FUNCTION_BLOCK UInterface EXTENDS OperationalParticleSet
  VAR CONSTANT
    cStartPeriod : t_ms_time := TIME#2s0ms;
  END_VAR
  VAR
    lVROverrideRadioReady : ValueReferenceBool;
    lOverrideRadioReady : BOOL := FALSE;
    lAlarmUInterfaceEstop : ReportableSystemControl;
    lAlarmUInterfaceStop : ReportableSystemControl;
    lAlarmUInterfaceEmgy : ReportableSystemControl;
    lAlarmUInterfaceNotReady : ReportableSystemControl;
    lUInterfaceId : t_ui_id := t_ui_id.cUIIdNone;
    lResolved : REFERENCE TO UInterface;
    lSingleMode : BOOL := TRUE;
    lUIMode : t_ui_mode := cUIModeInoperable;
    lUIModeRequest : BOOL := FALSE;
    lReady : BOOL := FALSE;
    lDiagnostic : t_uinterface_diagnostic;
    _Diagnostic : t_uinterface_diagnostic;
  END_VAR

            ;
          

METHOD operator
                  lDiagnostic := _Diagnostic;
_Diagnostic := cUInterfaceDiagnosticOK;

SUPER^.operator();

(* events for radios that are not present are ignored if in multi mode *)
IF (lSingleMode) THEN
	lUIMode := cUIModeSingle;
END_IF

IF ((NOT(Estop)) AND (lUIMode>cUIModeInoperable)) THEN
	Diagnostic := cUInterfaceDiagnosticEstop;

	lAlarmUInterfaceEstop.trigger(FALSE);
END_IF

IF ((NOT(Stop)) AND (lUIMode>cUIModeInoperable)) THEN
	Diagnostic := cUInterfaceDiagnosticStop;

	lAlarmUInterfaceStop.trigger(FALSE);
END_IF

IF ((NOT(Emgy)) AND (lUIMode>cUIModeInoperable))  THEN
	Diagnostic := cUInterfaceDiagnosticEmgy;

	lAlarmUInterfaceEmgy.trigger(FALSE);
END_IF

lReady := ((Stop) AND (Emgy) AND (Estop));
IF (NOT(Ready)) THEN
	lUIMode := cUIModeInoperable;

	IF (lSingleMode) THEN
		Diagnostic := cUInterfaceDiagnosticNotReady;
	
		lAlarmUInterfaceNotReady.trigger(FALSE);
	END_IF
END_IF

IF (UIModeResponse) THEN
	Resolved.uiModeHandler(UInterfaceId);
END_IF

IF (lUIMode=cUIModeInoperable) THEN
	Diagnostic := cUInterfaceDiagnosticInoperable;
	RETURN;
END_IF

IF (lUIMode<cUIModeMaster) THEN
	Diagnostic := cUInterfaceDiagnosticNotMaster;
	RETURN;
END_IF


                
END_METHOD

METHOD uiModeHandler
  VAR_INPUT
    id : t_ui_id;
  END_VAR
                  
                
END_METHOD

METHOD initialize
                  lResolved REF= THIS^;

lVROverrideRadioReady.initializeValueReference(lOverrideRadioReady,NopSelf,'OvrdReady','Override UI to be ready','',cValueStyleParameter);

lAlarmUInterfaceEstop.initializeState(NopSelf,'',cACUInterfaceEstop); // foobar life was zero
lAlarmUInterfaceEstop.Control := cSystemControlStop;
lAlarmUInterfaceEstop.AllowableSystemState := cSystemStateCharging;

lAlarmUInterfaceStop.initializeState(NopSelf,'',cACUInterfaceStop);
lAlarmUInterfaceStop.Control := cSystemControlStop;
lAlarmUInterfaceStop.AllowableSystemState := cSystemStateCharging;
		
lAlarmUInterfaceEmgy.initializeState(NopSelf,'',cACUInterfaceEmgy);
lAlarmUInterfaceEmgy.Control := cSystemControlStop;
lAlarmUInterfaceEmgy.AllowableSystemState := cSystemStateCharging;

lAlarmUInterfaceNotReady.initializeState(NopSelf,'',cACUInterfaceNotReady);
lAlarmUInterfaceNotReady.Control := cSystemControlStop;
lAlarmUInterfaceNotReady.AllowableSystemState := cSystemStateCharging;

SUPER^.initialize();
SubSystem := cSubsystemUInterface;

lReady := FALSE;
lUIMode := cUIModeInoperable;
//lInputMode := cInputModeDefault;
                
END_METHOD

PROPERTY LiftBalanceAB : t_percentage
GET
                    LiftBalanceAB := 0;
                  
END_GET
END_PROPERTY

PROPERTY LiftBalanceAD : t_percentage
GET
                    LiftBalanceAD := 0;
                  
END_GET
END_PROPERTY

(* {attribute 'monitoring' := 'call'} *)
PROPERTY LiftJoystickInputPresent : BOOL
GET
                    LiftJoystickInputPresent := false;

                  
END_GET
END_PROPERTY

PROPERTY OperatingMethodRequest : t_operating_method
GET
                    OperatingMethodRequest := cOperatingMethodNone;

                  
END_GET
END_PROPERTY

PROPERTY Override : BOOL
GET
                    Override := false;
                  
END_GET
END_PROPERTY

PROPERTY Present : BOOL
GET
                    Present := (UIMode>t_ui_mode.cUIModeInoperable);

                  
END_GET
END_PROPERTY

(* {attribute 'monitoring' := 'call'} *)
PROPERTY Ready : BOOL
GET
                    Ready := ((lReady) OR (lOverrideRadioReady));

                  
END_GET
END_PROPERTY

PROPERTY SideshiftAB : t_percentage
GET
                    SideshiftAB := 0;

                  
END_GET
END_PROPERTY

PROPERTY SideshiftCD : t_percentage
GET
                    SideshiftCD := 0;

                  
END_GET
END_PROPERTY

PROPERTY SingleMode : BOOL
GET
                    SingleMode := lSingleMode;
                  
END_GET
SET
                    lSingleMode := SingleMode;
                  
END_SET
END_PROPERTY

PROPERTY SlowFactor : REAL
GET
                    SlowFactor := 1.0;

                  
END_GET
END_PROPERTY

PROPERTY SpreaderTelescopingExtend : BOOL
GET
                    SpreaderTelescopingExtend := FALSE;

                  
END_GET
END_PROPERTY

PROPERTY SpreaderTelescopingRetract : BOOL
GET
                    SpreaderTelescopingRetract := FALSE;

                  
END_GET
END_PROPERTY

PROPERTY Steer : t_percentage
GET
                    Steer := 0;
                  
END_GET
END_PROPERTY

PROPERTY SteerModeRequest : t_steer_mode
GET
                    SteerModeRequest := cSteerModeNone;

                  
END_GET
END_PROPERTY

PROPERTY Stop : BOOL
GET
                    Stop := true;
                  
END_GET
END_PROPERTY

PROPERTY Topbeam : t_percentage
GET
                    Topbeam := 0;
                  
END_GET
END_PROPERTY

(* {attribute 'monitoring' := 'call'} *)
PROPERTY Travel : t_percentage
GET
                    Travel := 0;
                  
END_GET
END_PROPERTY

(* {attribute 'monitoring' := 'call'} *)
PROPERTY TravelJoystickInputPresent : BOOL
GET
                    TravelJoystickInputPresent := false;

                  
END_GET
END_PROPERTY

PROPERTY TwistlockLock : BOOL
GET
                    TwistlockLock := false;
                  
END_GET
END_PROPERTY

PROPERTY TwistlockUnlock : BOOL
GET
                    TwistlockUnlock := false;
                  
END_GET
END_PROPERTY

PROPERTY TypeToken : t_medium_string
GET
                    TypeToken := 'UInterface';
                  
END_GET
END_PROPERTY

PROPERTY UIEventCodeRequest : t_ui_event_code
GET
                    UIEventCodeRequest := cUIEventCodeNone;
                  
END_GET
END_PROPERTY

(* {attribute 'monitoring' := 'call'} *)
PROPERTY UIMode : t_ui_mode
GET
                    UIMode := lUIMode;

                  
END_GET
SET
                    lUIMode := UIMode;
                  
END_SET
END_PROPERTY

(* {attribute 'monitoring' := 'call'} *)
PROPERTY UIModeRequest : BOOL
GET
                    UIModeRequest := lUIModeRequest;
                  
END_GET
SET
                    lUIModeRequest := UIModeRequest;
                  
END_SET
END_PROPERTY

(* {attribute 'monitoring' := 'call'} *)
PROPERTY UIModeResponse : BOOL
GET
                    UIModeResponse := FALSE;


                  
END_GET
END_PROPERTY

PROPERTY UInterfaceId : t_ui_id
GET
                    UInterfaceId := lUInterfaceId;
                  
END_GET
SET
                    lUInterfaceId := UInterfaceId;
                  
END_SET
END_PROPERTY

PROPERTY UIOrientation : t_ui_orientation
GET
                    UIOrientation := cUIOrientationForward;
                  
END_GET
END_PROPERTY

PROPERTY UMFS : BOOL
GET
                    UMFS := true;
                  
END_GET
END_PROPERTY

PROPERTY ZeroSteerTargetAngle : BOOL
GET
                    ZeroSteerTargetAngle := false;
                  
END_GET
END_PROPERTY

PROPERTY Resolved : REFERENCE TO UInterface
GET
                    Resolved ref= lResolved;
                  
END_GET
SET
                    lResolved ref= Resolved;
                  
END_SET
END_PROPERTY

PROPERTY Active : BOOL
GET
                    Active := (UIMode>cUIModeSlave);

                  
END_GET
END_PROPERTY

PROPERTY AutomationRequest : t_prog_mov_code
GET
                    AutomationRequest := cProgMovCodeNone;
                  
END_GET
END_PROPERTY

PROPERTY AutomationStart : BOOL
GET
                    AutomationStart := FALSE;

                  
END_GET
END_PROPERTY

(* {attribute 'monitoring' := 'call'} *)
PROPERTY ConfigurationJoystickInputPresent : BOOL
GET
                    ConfigurationJoystickInputPresent := FALSE;

                  
END_GET
END_PROPERTY

PROPERTY Diagnostic : t_uinterface_diagnostic
GET
                    Diagnostic := lDiagnostic;
                  
END_GET
SET
                    _Diagnostic := Diagnostic;
                  
END_SET
END_PROPERTY

PROPERTY Emgy : BOOL
GET
                    Emgy := true;
                  
END_GET
END_PROPERTY

PROPERTY Estop : BOOL
GET
                    Estop := true;
                  
END_GET
END_PROPERTY

PROPERTY FunctionalModeRequest : t_functional_mode
GET
                    FunctionalModeRequest := cFunctionalModeAny;

                  
END_GET
END_PROPERTY

PROPERTY Horn : BOOL
GET
                    Horn := false;
                  
END_GET
END_PROPERTY

PROPERTY InputMode : t_input_mode
GET
                    InputMode := cInputModeDefault;

                  
END_GET
END_PROPERTY

PROPERTY IsBeginner : BOOL
GET
                    IsBeginner := FALSE;

                  
END_GET
END_PROPERTY

PROPERTY IsSlow : BOOL
GET
                    IsSlow := FALSE;

                  
END_GET
END_PROPERTY

(* {attribute 'monitoring' := 'call'} *)
PROPERTY JoystickInputPresent : BOOL
GET
                    JoystickInputPresent := false;
                  
END_GET
END_PROPERTY

PROPERTY Lift : t_percentage
GET
                    Lift := 0;
                  
END_GET
END_PROPERTY

PROPERTY EnableBatteryPack : BOOL
GET
                    EnableBatteryPack := FALSE;

                  
END_GET
END_PROPERTY
END_FUNCTION_BLOCK

FUNCTION_BLOCK ExtractTest
  VAR
    mWordA : WORD;
    mWordB : WORD;
    mWordC : WORD;
    mWordD : WORD;
    mBoolA : BOOL;
    mBoolB : BOOL;
    mBoolC : BOOL;
    mIntA : INT;
    mIntB : INT;
    mIntC : INT;
    mIntD : INT;
    mByteA : BYTE;
    mByteB : BYTE;
    mByteC : BYTE;
    mByteD : BYTE;
    mStartA : USINT := 0;
    mStartB : USINT := 0;
    mStartC : USINT := 0;
    mStartD : USINT := 0;
    mStartE : USINT := 0;
    mStartF : USINT := 0;
    mLengthA : USINT := 0;
    mLengthB : USINT := 0;
  END_VAR

            mByteA := fInsertBool(pData:=mBoolA,pStart:=mStartA);
mByteB := fInsertBits(pData:=mIntA,pStart:=mStartB);
mByteC := fMergeBits(pByte:=mByteA,pData:=mIntB,pStart:=mStartC);

mWordA := fInsertBoolIntoWord(pData:=mBoolA,pStart:=mStartD);
mWordB := fInsertBitsIntoWord(pData:=mIntA,pStart:=mStartE);
mWordC := fMergeBitsIntoWord(pWord:=mWordA,pData:=mIntB,pStart:=mStartF);

mBoolB := fExtractBool(pByte:=mByteA,pStart:=mStartA);
mBoolC := fExtractBoolFromWord(pWord:=mWordA,pStart:=mStartD);

mIntC := fExtractBits(pByte:=mByteB,pStart:=mStartB,pLength:=mLengthA);
mIntD := fExtractBitsFromWord(pWord:=mWordB,pStart:=mStartE,pLength:=mLengthB);

mWordD :=  fExtractWord(pByte1:=mByteA ,pByte2:=mByteB);
          
END_FUNCTION_BLOCK

FUNCTION fExtractBits : INT
  VAR_INPUT
    pByte : BYTE;
    pStart : USINT;
    pLength : USINT;
  END_VAR

            fExtractBits := SHR(SHL(pByte,8-pStart-pLength),8-pLength);
          
END_FUNCTION

FUNCTION fExtractBitsFromWord : INT
  VAR_INPUT
    pWord : WORD;
    pStart : USINT;
    pLength : USINT;
  END_VAR

            fExtractBitsFromWord := WORD_TO_INT(SHR(SHL(pWord,16-pStart-pLength),16-pLength));
          
END_FUNCTION

FUNCTION fExtractBool : BOOL
  VAR_INPUT
    pByte : BYTE;
    pStart : USINT;
  END_VAR

            fExtractBool := BYTE_TO_BOOL(pByte AND SHL(BOOL_TO_BYTE(TRUE),pStart));
          
END_FUNCTION

FUNCTION fExtractBoolFromWord : BOOL
  VAR_INPUT
    pWord : WORD;
    pStart : USINT;
  END_VAR

            fExtractBoolFromWord := WORD_TO_BOOL(pWord AND SHL(BOOL_TO_WORD(TRUE),pStart));
          
END_FUNCTION

FUNCTION fExtractWord : WORD
  VAR_INPUT
    pByte1 : BYTE;
    pByte2 : BYTE;
  END_VAR

            fExtractWord := SHL(BYTE_TO_WORD(pByte2),8) OR BYTE_TO_WORD(pByte1);
          
END_FUNCTION

FUNCTION fInsertBits : BYTE
  VAR_INPUT
    pData : INT;
    pStart : USINT;
  END_VAR

            fInsertBits := SHL(INT_TO_BYTE(pData),pStart);
          
END_FUNCTION

FUNCTION fInsertBitsIntoWord : WORD
  VAR_INPUT
    pData : INT;
    pStart : USINT;
  END_VAR

            fInsertBitsIntoWord := SHL(INT_TO_WORD(pData),pStart);
          
END_FUNCTION

FUNCTION fInsertBool : BYTE
  VAR_INPUT
    pData : BOOL;
    pStart : USINT;
  END_VAR

            fInsertBool := SHL(BOOL_TO_BYTE(pData),pStart);
          
END_FUNCTION

FUNCTION fInsertBoolIntoWord : WORD
  VAR_INPUT
    pData : BOOL;
    pStart : USINT;
  END_VAR

            fInsertBoolIntoWord := SHL(BOOL_TO_WORD(pData),pStart);
          
END_FUNCTION

FUNCTION fMergeBits : BYTE
  VAR_INPUT
    pByte : BYTE;
    pData : INT;
    pStart : USINT;
  END_VAR

            fMergeBits := SHL(INT_TO_BYTE(pData),pStart) OR (pByte);
          
END_FUNCTION

FUNCTION fMergeBitsIntoBytes : WORD
  VAR_INPUT
    pByte1 : BYTE;
    pByte2 : BYTE;
    pData : INT;
    pStart : USINT;
  END_VAR

            fMergeBitsIntoBytes := SHL(INT_TO_WORD(pData),pStart) OR (SHL(BYTE_TO_WORD(pByte2),8) OR BYTE_TO_WORD(pByte1));
          
END_FUNCTION

FUNCTION fMergeBitsIntoWord : WORD
  VAR_INPUT
    pWord : WORD;
    pData : INT;
    pStart : USINT;
  END_VAR

            fMergeBitsIntoWord := SHL(INT_TO_WORD(pData),pStart) OR (pWord);
          
END_FUNCTION

FUNCTION fMergeBool : BYTE
  VAR_INPUT
    pByte : BYTE;
    pData : BOOL;
    pStart : USINT;
  END_VAR

            fMergeBool := SHL(BOOL_TO_BYTE(pData),pStart) OR (pByte);
          
END_FUNCTION

FUNCTION fMergeBoolIntoWord : WORD
  VAR_INPUT
    pWord : WORD;
    pData : BOOL;
    pStart : USINT;
  END_VAR

            fMergeBoolIntoWord := SHL(BOOL_TO_WORD(pData),pStart) OR (pWord);
          
END_FUNCTION

FUNCTION_BLOCK ValueObjectBoolChange EXTENDS ValueObjectBool
  VAR
    lPreviousValue : BOOL;
    lRising : BOOL := FALSE;
    lFalling : BOOL := FALSE;
  END_VAR

            
          

METHOD operator
                  SUPER^.operator();

lFalling := ((NOT(Value)) AND (lPreviousValue));
lRising := ((Value) AND (NOT(lPreviousValue)));

lPreviousValue := Value;

                
END_METHOD

(* {attribute 'monitoring' := 'call'} *)
PROPERTY Falling : BOOL
GET
                    Falling := lFalling;
                  
END_GET
END_PROPERTY

(* {attribute 'monitoring' := 'call'} *)
PROPERTY Rising : BOOL
GET
                    Rising := lRising;
                  
END_GET
END_PROPERTY
END_FUNCTION_BLOCK

FUNCTION_BLOCK ValueObjectBoolCheckReferenceDINT EXTENDS ValueObjectBool
  VAR
    lCheckReference : REFERENCE TO DINT;
    _CheckReference : DINT;
    lTimer : t_timer;
    lCheckRequiredValue : BOOL := TRUE;
    lCheckEnable : BOOL := TRUE;
    lCheckCritical : BOOL := FALSE;
    lError : BOOL := FALSE;
    lPrevious : BOOL;
    lChanged : BOOL;
    lOK : BOOL;
    lOKOff : BOOL;
    lOff : BOOL;
  END_VAR

            
          

METHOD initialize
                  IF (NOT(__ISVALIDREF(lCheckReference))) THEN
	lCheckReference REF= _CheckReference;
END_IF

_CheckReference := 0;

SUPER^.initialize();

lTimer.initialize();
lTimer.Enable := true;

lValue := lPrevious := lError := lOK := lOKOff := lOff := lChanged := FALSE;

                
END_METHOD

METHOD operator
                  IF (lPrevious<>lValue) THEN
	lChanged := TRUE;
	lPrevious := lValue;
	lTimer.reset();
ELSE
	lChanged := FALSE;
END_IF

SUPER^.operator();

lTimer.operator();

lError := ((lTimer.lExpired) AND
	(lValue) AND
	(lCheckEnable) AND
	(DINT_TO_BOOL(lCheckReference)<>lCheckRequiredValue));	

(* waits to set OK until timer has expired *)
lOK :=  ((lTimer.lExpired) AND (lValue) AND (NOT(lError)));
lOKOff :=  ((lTimer.lExpired) AND (NOT(lValue)) AND (NOT(lError)));
lOff := ((lTimer.lExpired) AND (NOT(lValue)));


                
END_METHOD

PROPERTY CheckCritical : BOOL
GET
                    CheckCritical := lCheckCritical;
                  
END_GET
SET
                    lCheckCritical := CheckCritical;
                  
END_SET
END_PROPERTY

PROPERTY CheckEnable : BOOL
GET
                    CheckEnable := lCheckEnable;
                  
END_GET
SET
                    lCheckEnable := CheckEnable;
                  
END_SET
END_PROPERTY

PROPERTY CheckPeriod : t_time
GET
                    CheckPeriod := lTimer.Period;
                  
END_GET
SET
                    lTimer.Period := CheckPeriod;

                  
END_SET
END_PROPERTY

PROPERTY Error : BOOL
GET
                    Error := lError;
                  
END_GET
END_PROPERTY

PROPERTY IsOff : BOOL
GET
                    IsOff := lOff;
                  
END_GET
END_PROPERTY

PROPERTY OK : BOOL
GET
                    OK := lOK;
                  
END_GET
END_PROPERTY

PROPERTY OKOff : BOOL
GET
                    OKOff := lOKOff;
                  
END_GET
END_PROPERTY

PROPERTY CheckReference : REFERENCE TO DINT
SET
                    lCheckReference Ref= CheckReference;
                  
END_SET
END_PROPERTY
END_FUNCTION_BLOCK

FUNCTION_BLOCK ValueObjectBoolCheckReferenceDINTOutputReferenceDINT EXTENDS ValueObjectBoolCheckReferenceDINT
  VAR
    lOutputReference : REFERENCE TO DINT;
  END_VAR

            
          

METHOD operator
                  SUPER^.operator();

lOutputReference := BOOL_TO_DINT(lValue);
                
END_METHOD

METHOD initialize
                  IF (NOT(__ISVALIDREF(lOutputReference))) THEN
	gCodeErrorHandler(pMessage:=CONCAT('null reference in ',lIdentity));
END_IF

SUPER^.initialize();

                
END_METHOD

PROPERTY OutputReference : REFERENCE TO DINT
SET
                    lOutputReference ref= OutputReference;
                  
END_SET
END_PROPERTY
END_FUNCTION_BLOCK

FUNCTION_BLOCK ValueObjectBoolInputRealThreshold EXTENDS ValueObjectBool
  VAR
    lInput : REAL;
    lBelowIsOn : BOOL;
    lThresholdOn : REAL;
    lThresholdOff : REAL;
    lHysteresis : REAL := 2.0;
    lThreshold : REAL := 30.0;
  END_VAR

            
          

METHOD operator
                  IF (lBelowIsOn) THEN
	// generally lThresholdBelowIsOn (off->on) < lThresholdLowerOff (on->off)
	IF ((lInput<=lThresholdOn) OR
		((lValue) AND (lInput<=lThresholdOff))) THEN
		lValue := TRUE;
	ELSE
		lValue := FALSE;
	END_IF
ELSE
	// generally lThresholdUpperOn (off->on) > lThresholdUpperOff (on->off)
	IF ((lInput>=lThresholdOn) OR
		((lValue) AND (lInput>=lThresholdOff))) THEN
		lValue := TRUE;
	ELSE
		lValue := FALSE;
	END_IF
END_IF

SUPER^.operator();


                
END_METHOD

METHOD describe
  VAR_INPUT
    executeContext : POINTER TO ExecuteContext;
  END_VAR
                  SUPER^.describe(executeContext);

IF (executeContext^.matchOption(cExecuteOptionSyntax)) THEN
	executeContext^.describeSyntaxConfigurable(lStyle,cTokenThreshold,cDataTypeReal,cEnumTypeNone,lUnits,cDescriptionThreshold);
	executeContext^.describeSyntaxConfigurable(lStyle,cTokenHysteresis,cDataTypeReal,cEnumTypeNone,lUnits,cDescriptionHysteresis);
	
	RETURN;
END_IF

IF (executeContext^.matchOption(cExecuteOptionParameter)) THEN
	executeContext^.describeParameter(lStyle,lIdentity,cTokenThreshold,gTypeHandler.getTokenForReal(lThreshold),cDataTypeReal,cEnumTypeNone,lUnits,cDescriptionThreshold);
	executeContext^.describeParameter(cValueStyleParameter,lIdentity,cTokenHysteresis,gTypeHandler.getTokenForReal(lHysteresis),cDataTypeReal,cEnumTypeNone,lUnits,cDescriptionHysteresis);
		
	RETURN;
END_IF

executeContext^.appendTokenPair(cTokenThreshold,gTypeHandler.getTokenForReal(lThreshold),FALSE,TRUE);
executeContext^.appendTokenPair(cTokenHysteresis,gTypeHandler.getTokenForReal(lHysteresis),FALSE,TRUE);
executeContext^.appendTokenPair(cTokenHysteresis,gTypeHandler.getTokenForUSINT(BOOL_TO_USINT(lBelowIsOn)),FALSE,TRUE);




                
END_METHOD

METHOD configure
  VAR_INPUT
    executeContext : POINTER TO ExecuteContext;
  END_VAR
                  IF (executeContext^.configureReal(cTokenThreshold,lThreshold,FALSE,THIS)) THEN
	RETURN;
END_IF

IF (executeContext^.configureReal(cTokenHysteresis,lHysteresis,FALSE,THIS)) THEN
	RETURN;
END_IF

SUPER^.configure(executeContext);


                
END_METHOD

METHOD setThresholds : BOOL
                  IF (lBelowIsOn) THEN
	lThresholdOff := Threshold + lHysteresis;
	lThresholdOn := Threshold - lHysteresis;
ELSE
	lThresholdOff := Threshold - lHysteresis;
	lThresholdOn := Threshold + lHysteresis;	
END_IF
                
END_METHOD

METHOD initialize
                  SUPER^.initialize();

setThresholds();
                
END_METHOD

PROPERTY Input : REAL
SET
                    lInput := Input;
operator();

                  
END_SET
END_PROPERTY

PROPERTY ThresholdOff : REAL
GET
                    ThresholdOff := lThresholdOff;
                  
END_GET
END_PROPERTY

PROPERTY ThresholdOn : REAL
GET
                    ThresholdOn := ThresholdOn;
                  
END_GET
END_PROPERTY

PROPERTY Hysteresis : REAL
GET
                    Hysteresis := lHysteresis;
                  
END_GET
SET
                    IF (lHysteresis=Hysteresis) THEN
	RETURN;
END_IF

lHysteresis := Hysteresis;
setThresholds();
                  
END_SET
END_PROPERTY

PROPERTY Threshold : REAL
GET
                    Threshold := lThreshold;
                  
END_GET
SET
                    IF (lThreshold=Threshold) THEN
	RETURN;
END_IF

lThreshold := Threshold;
setThresholds();
                  
END_SET
END_PROPERTY

PROPERTY BelowIsOn : BOOL
GET
                    BelowIsOn := lBelowIsOn;
                  
END_GET
SET
                    lBelowIsOn := BelowIsOn;
setThresholds();

                  
END_SET
END_PROPERTY
END_FUNCTION_BLOCK

FUNCTION_BLOCK ValueObjectBoolInputReferenceBool EXTENDS ValueObjectBool
  VAR
    lInputReference : REFERENCE TO BOOL;
  END_VAR

            
          

METHOD initialize
                  IF (NOT(__ISVALIDREF(lInputReference))) THEN
	gCodeErrorHandler(pMessage:=CONCAT('null reference in ',lIdentity));
END_IF

SUPER^.initialize();

                
END_METHOD

METHOD operator
                  lValue := lInputReference;

SUPER^.operator();

                
END_METHOD

PROPERTY InputReference : REFERENCE TO BOOL
SET
                    lInputReference REF= InputReference;


                  
END_SET
END_PROPERTY
END_FUNCTION_BLOCK

FUNCTION_BLOCK ValueObjectBoolInputReferenceBoolAndBool EXTENDS ValueObjectBool
  VAR
    lInputReferenceA : REFERENCE TO BOOL;
    lInputReferenceB : REFERENCE TO BOOL;
  END_VAR

            
          

METHOD initialize
                  IF ((NOT(__ISVALIDREF(lInputReferenceA))) OR
	(NOT(__ISVALIDREF(lInputReferenceB)))) THEN
	gCodeErrorHandler(pMessage:=CONCAT('null reference in ',lIdentity));
END_IF

SUPER^.initialize();

                
END_METHOD

METHOD operator
                  lValue := ((lInputReferenceA) AND (lInputReferenceB));

SUPER^.operator();

                
END_METHOD

PROPERTY InputReferenceA : REFERENCE TO BOOL
SET
                    lInputReferenceA REF= InputReferenceA;


                  
END_SET
END_PROPERTY

PROPERTY InputReferenceB : REFERENCE TO BOOL
SET
                    lInputReferenceB REF= InputReferenceB;


                  
END_SET
END_PROPERTY
END_FUNCTION_BLOCK

FUNCTION_BLOCK ValueObjectBoolInputReferenceBoolChange EXTENDS ValueObjectBool
  VAR
    lInputReference : REFERENCE TO BOOL;
    lPreviousValue : BOOL;
    lRising : BOOL := FALSE;
    lFalling : BOOL := FALSE;
  END_VAR

            
          

METHOD operator
                  lValue := lInputReference;

SUPER^.operator();

lFalling := ((NOT(Value)) AND (lPreviousValue));
lRising := ((Value) AND (NOT(lPreviousValue)));

lPreviousValue := Value;

                
END_METHOD

METHOD initialize
                  IF (NOT(__ISVALIDREF(lInputReference))) THEN
	gCodeErrorHandler(pMessage:=CONCAT('null reference in ',lIdentity));
END_IF

SUPER^.initialize();

                
END_METHOD

(* {attribute 'monitoring' := 'call'} *)
PROPERTY Falling : BOOL
GET
                    Falling := lFalling;
                  
END_GET
END_PROPERTY

(* {attribute 'monitoring' := 'call'} *)
PROPERTY Rising : BOOL
GET
                    Rising := lRising;
                  
END_GET
END_PROPERTY

PROPERTY InputReference : REFERENCE TO BOOL
SET
                    lInputReference REF= InputReference;


                  
END_SET
END_PROPERTY
END_FUNCTION_BLOCK

FUNCTION_BLOCK ValueObjectBoolInputReferenceDINTAsBool EXTENDS ValueObjectBool
  VAR
    lInputReference : REFERENCE TO DINT;
  END_VAR

            
          

METHOD initialize
                  IF (NOT(__ISVALIDREF(lInputReference))) THEN
	gCodeErrorHandler(pMessage:=CONCAT('null reference in ',lIdentity));
END_IF

SUPER^.initialize();

                
END_METHOD

METHOD operator
                  lValue := DINT_TO_BOOL(lInputReference);

SUPER^.operator();

                
END_METHOD

PROPERTY InputReference : REFERENCE TO DINT
SET
                    lInputReference REF= InputReference;


                  
END_SET
END_PROPERTY
END_FUNCTION_BLOCK

FUNCTION_BLOCK ValueObjectBoolInputReferenceDINTFiltered EXTENDS ValueObjectBool
  VAR
    lInputReference : REFERENCE TO DINT;
    lFilterEnabled : BOOL := TRUE;
    lPrevious : BOOL;
    lTimer : t_timer;
  END_VAR

            
          

METHOD initialize
                  IF (NOT(__ISVALIDREF(lInputReference))) THEN
	gCodeErrorHandler(pMessage:=CONCAT('null reference in ',lIdentity));
END_IF

SUPER^.initialize();

lTimer.initialize();
lTimer.Enable := TRUE;
lTImer.Period := T#100MS;

lPrevious := lValue;

                
END_METHOD

METHOD operator
                  IF (lFilterEnabled) THEN
	IF (lPrevious<>DINT_TO_BOOL(lInputReference)) THEN
		lTimer.reset();
	END_IF

	lTimer.operator();
	IF (lTimer.Expired) THEN
		lValue := DINT_TO_BOOL(lInputReference);
	END_IF
ELSE
	lValue := DINT_TO_BOOL(lInputReference);
END_IF

lPrevious := DINT_TO_BOOL(lInputReference);

SUPER^.operator();

                
END_METHOD

PROPERTY FilterEnabled : BOOL
GET
                    FilterEnabled := lFilterEnabled;
                  
END_GET
SET
                    lFilterEnabled := FilterEnabled;
                  
END_SET
END_PROPERTY

PROPERTY Period : t_time
GET
                    Period := lTimer.Period;
                  
END_GET
SET
                    lTimer.Period := Period;
                  
END_SET
END_PROPERTY

PROPERTY InputReference : REFERENCE TO DINT
SET
                    lInputReference REF= InputReference;


                  
END_SET
END_PROPERTY
END_FUNCTION_BLOCK

FUNCTION_BLOCK ValueObjectBoolInputReferenceUINT EXTENDS ValueObjectBool
  VAR
    lInputReference : REFERENCE TO UINT;
    lIndex : USINT;
  END_VAR

            
          

METHOD initialize
                  IF (NOT(__ISVALIDREF(lInputReference))) THEN
	gCodeErrorHandler(pMessage:=CONCAT('null reference in ',lIdentity));
END_IF

SUPER^.initialize();

                
END_METHOD

METHOD operator
                  lValue := fExtractBoolFromWord(UINT_TO_WORD(lInputReference),pStart:=lIndex);

SUPER^.operator();

                
END_METHOD

PROPERTY Index : USINT
GET
                    Index := lIndex;
                  
END_GET
SET
                    lIndex := MIN(Index,15);
                  
END_SET
END_PROPERTY

PROPERTY InputReference : REFERENCE TO UINT
SET
                    lInputReference REF= InputReference;


                  
END_SET
END_PROPERTY
END_FUNCTION_BLOCK

FUNCTION_BLOCK ValueObjectBoolInputReferenceUSINT EXTENDS ValueObjectBool
  VAR
    lInputReference : REFERENCE TO USINT;
    lIndex : USINT;
  END_VAR

            
          

METHOD initialize
                  IF (NOT(__ISVALIDREF(lInputReference))) THEN
	gCodeErrorHandler(pMessage:=CONCAT('null reference in ',lIdentity));
END_IF

SUPER^.initialize();

                
END_METHOD

METHOD operator
                  lValue := fExtractBoolFromWord(USINT_TO_WORD(lInputReference),pStart:=lIndex);

SUPER^.operator();

                
END_METHOD

PROPERTY Index : USINT
GET
                    Index := lIndex;
                  
END_GET
SET
                    lIndex := MIN(Index,7);
                  
END_SET
END_PROPERTY

PROPERTY InputReference : REFERENCE TO USINT
SET
                    lInputReference REF= InputReference;


                  
END_SET
END_PROPERTY
END_FUNCTION_BLOCK

FUNCTION_BLOCK ValueObjectBoolInputReferenceUSINTAsBool EXTENDS ValueObjectBool
  VAR
    lInputReference : REFERENCE TO USINT;
  END_VAR

            
          

METHOD initialize
                  IF (NOT(__ISVALIDREF(lInputReference))) THEN
	gCodeErrorHandler(pMessage:=CONCAT('null reference in ',lIdentity));
END_IF

SUPER^.initialize();

                
END_METHOD

METHOD operator
                  lValue := USINT_TO_BOOL(lInputReference);

SUPER^.operator();

                
END_METHOD

PROPERTY InputReference : REFERENCE TO USINT
SET
                    lInputReference REF= InputReference;


                  
END_SET
END_PROPERTY
END_FUNCTION_BLOCK

FUNCTION_BLOCK ValueObjectBoolInputReferenceUSINTChange EXTENDS ValueObjectBoolChange
  VAR
    lInputReference : REFERENCE TO USINT;
    lIndex : USINT;
  END_VAR

            
          

METHOD operator
                  lValue := fExtractBoolFromWord(USINT_TO_WORD(lInputReference),pStart:=lIndex);

SUPER^.operator();

lPreviousValue := Value;

                
END_METHOD

METHOD initialize
                  IF (NOT(__ISVALIDREF(lInputReference))) THEN
	gCodeErrorHandler(pMessage:=CONCAT('null reference in ',lIdentity));
END_IF

SUPER^.initialize();

                
END_METHOD

PROPERTY InputReference : REFERENCE TO USINT
SET
                    lInputReference REF= InputReference;


                  
END_SET
END_PROPERTY

PROPERTY Index : USINT
GET
                    Index := lIndex;
                  
END_GET
SET
                    lIndex := MIN(Index,7);
                  
END_SET
END_PROPERTY
END_FUNCTION_BLOCK

FUNCTION_BLOCK ValueObjectBoolLatch EXTENDS ValueObjectBoolChange

            
          

METHOD reset
                  lValue := FALSE;
operator();
                
END_METHOD

PROPERTY Input : BOOL
SET
                    IF (Input) THEN
	lValue := Input;
END_IF

operator();

                  
END_SET
END_PROPERTY
END_FUNCTION_BLOCK

FUNCTION_BLOCK ValueObjectBoolOutputReferenceBool EXTENDS ValueObjectBool
  VAR
    lOutputReference : REFERENCE TO BOOL;
  END_VAR

            
          

METHOD operator
                  SUPER^.operator();

lOutputReference := lValue;


                
END_METHOD

METHOD initialize
                  IF (NOT(__ISVALIDREF(lOutputReference))) THEN
	gCodeErrorHandler(pMessage:=CONCAT('null reference in ',lIdentity));
END_IF

SUPER^.initialize();

                
END_METHOD

PROPERTY OutputReference : REFERENCE TO BOOL
SET
                    lOutputReference ref= OutputReference;
                  
END_SET
END_PROPERTY
END_FUNCTION_BLOCK

FUNCTION_BLOCK ValueObjectBoolOutputReferenceDINTAsBool EXTENDS ValueObjectBool
  VAR
    _Output : DINT;
    lOutputReference : REFERENCE TO DINT := _Output;
    lScaling : DINT := 1;
  END_VAR

            
          

METHOD operator
                  SUPER^.operator();

lOutputReference := BOOL_TO_DINT(lValue);


                
END_METHOD

METHOD initialize
                  IF (NOT(__ISVALIDREF(lOutputReference))) THEN
	gCodeErrorHandler(pMessage:=CONCAT('null reference in ',lIdentity));
END_IF

SUPER^.initialize();

                
END_METHOD

PROPERTY OutputReference : REFERENCE TO DINT
SET
                    lOutputReference ref= OutputReference;
                  
END_SET
END_PROPERTY
END_FUNCTION_BLOCK

FUNCTION_BLOCK ValueObjectBoolOutputReferenceDINTAsBoolOpt EXTENDS ValueObjectBool
  VAR
    _Output : DINT;
    lOutputReference : REFERENCE TO DINT := _Output;
    lScaling : DINT := 1;
  END_VAR

            
          

METHOD operator
                  SUPER^.operator();

lOutputReference := BOOL_TO_DINT(lValue)*lScaling;


                
END_METHOD

METHOD initialize
                  IF (NOT(__ISVALIDREF(lOutputReference))) THEN
	gCodeErrorHandler(pMessage:=CONCAT('null reference in ',lIdentity));
END_IF

SUPER^.initialize();

                
END_METHOD

PROPERTY Scaling : DINT
GET
                    Scaling := lScaling;
                  
END_GET
SET
                    lScaling := Scaling;
                  
END_SET
END_PROPERTY

PROPERTY OutputReference : REFERENCE TO DINT
SET
                    lOutputReference ref= OutputReference;
                  
END_SET
END_PROPERTY
END_FUNCTION_BLOCK

FUNCTION_BLOCK ValueObjectBoolOutputReferenceUSINT EXTENDS ValueObjectBool
  VAR
    lOutputReference : REFERENCE TO USINT;
    lIndex : USINT;
    lMergeOutput : BOOL := FALSE;
  END_VAR

            
          

METHOD operator
                  SUPER^.operator();

IF (lMergeOutput) THEN
	lOutputReference := fMergeBool(lOutputReference,lValue,pStart:=lIndex);
ELSE
	lOutputReference := fInsertBool(lValue,pStart:=lIndex);	
END_IF

                
END_METHOD

METHOD initialize
                  IF (NOT(__ISVALIDREF(lOutputReference))) THEN
	gCodeErrorHandler(pMessage:=CONCAT('null reference in ',lIdentity));
END_IF

SUPER^.initialize();

                
END_METHOD

PROPERTY OutputReference : REFERENCE TO USINT
SET
                    lOutputReference ref= OutputReference;
                  
END_SET
END_PROPERTY

PROPERTY Index : USINT
GET
                    Index := lIndex;
                  
END_GET
SET
                    lIndex := MIN(Index,7);
                  
END_SET
END_PROPERTY

PROPERTY MergeOutput : BOOL
GET
                    MergeOutput := lMergeOutput;
                  
END_GET
SET
                    lMergeOutput := MergeOutput;
                  
END_SET
END_PROPERTY
END_FUNCTION_BLOCK

FUNCTION_BLOCK ValueObjectBoolOutputReferenceUSINTAsBool EXTENDS ValueObjectBool
  VAR
    lOutputReference : REFERENCE TO USINT;
  END_VAR

            
          

METHOD operator
                  SUPER^.operator();

IF (lValue) THEN
	lOutputReference := 1;
ELSE
	lOutputReference := 0;
END_IF

                
END_METHOD

METHOD initialize
                  IF (NOT(__ISVALIDREF(lOutputReference))) THEN
	gCodeErrorHandler(pMessage:=CONCAT('null reference in ',lIdentity));
END_IF

SUPER^.initialize();

                
END_METHOD

PROPERTY OutputReference : REFERENCE TO USINT
SET
                    lOutputReference ref= OutputReference;
                  
END_SET
END_PROPERTY
END_FUNCTION_BLOCK

FUNCTION_BLOCK ValueObjectBoolOutputReferenceUSINTUSINT EXTENDS ValueObjectBool
  VAR
    lOutputReferenceA : REFERENCE TO USINT;
    lOutputReferenceB : REFERENCE TO USINT;
    lIndexA : USINT := 0;
    lIndexB : USINT := 0;
    lMergeOutputA : BOOL := FALSE;
    lMergeOutputB : BOOL := TRUE;
  END_VAR

            
          

METHOD operator
                  SUPER^.operator();

IF (lMergeOutputA) THEN
	lOutputReferenceA := fMergeBool(lOutputReferenceA,lValue,pStart:=lIndexA);
ELSE
	lOutputReferenceA := fInsertBool(lValue,pStart:=lIndexA);	
END_IF

IF (lMergeOutputB) THEN
	lOutputReferenceB := fMergeBool(lOutputReferenceB,lValue,pStart:=lIndexB);
ELSE
	lOutputReferenceB := fInsertBool(lValue,pStart:=lIndexB);	
END_IF



                
END_METHOD

METHOD initialize
                  IF ((NOT(__ISVALIDREF(lOutputReferenceA))) OR
	(NOT(__ISVALIDREF(lOutputReferenceB)))) THEN
	gCodeErrorHandler(pMessage:=CONCAT('null reference in ',lIdentity));
END_IF

SUPER^.initialize();

                
END_METHOD

PROPERTY OutputReferenceA : REFERENCE TO USINT
SET
                    lOutputReferenceA ref= OutputReferenceA;
                  
END_SET
END_PROPERTY

PROPERTY OutputReferenceB : REFERENCE TO USINT
SET
                    lOutputReferenceB ref= OutputReferenceB;
                  
END_SET
END_PROPERTY

PROPERTY IndexA : USINT
GET
                    IndexA := lIndexA;
                  
END_GET
SET
                    lIndexA := MIN(IndexA,7);
                  
END_SET
END_PROPERTY

PROPERTY IndexB : USINT
GET
                    IndexB := lIndexB;
                  
END_GET
SET
                    lIndexB := MIN(IndexB,7);
                  
END_SET
END_PROPERTY

PROPERTY MergeOutputA : BOOL
GET
                    MergeOutputA := lMergeOutputA;
                  
END_GET
SET
                    lMergeOutputA := MergeOutputA;
                  
END_SET
END_PROPERTY

PROPERTY MergeOutputB : BOOL
GET
                    MergeOutputB := lMergeOutputB;
                  
END_GET
SET
                    lMergeOutputB := MergeOutputB;
                  
END_SET
END_PROPERTY
END_FUNCTION_BLOCK

FUNCTION_BLOCK ValueObjectBoolOutputUINT EXTENDS ValueObjectBool
  VAR
    lOutput : UINT;
    lIndex : USINT;
  END_VAR

            
          

METHOD operator
                  SUPER^.operator();

lOutput := fInsertBool(lValue,pStart:=lIndex);

                
END_METHOD

PROPERTY Index : USINT
GET
                    Index := lIndex;
                  
END_GET
SET
                    lIndex := MIN(Index,15);
                  
END_SET
END_PROPERTY

PROPERTY Output : UINT
GET
                    operator();
Output := lOutput;

                  
END_GET
END_PROPERTY
END_FUNCTION_BLOCK

FUNCTION_BLOCK ValueObjectBoolParsedBool EXTENDS ValueObjectBool
  VAR
    lInput : BOOL;
    lPreviousInput : BOOL;
    lChanged : BOOL;
    lTriggerOnFalling : BOOL := FALSE;
    lTimer : t_timer;
    lDuration : t_ms_time;
    lExpired : BOOL;
    lExpiredTriggered : BOOL;
    lExpiredEvent : BOOL;
    lFastEvent : BOOL;
    lRising : BOOL;
    lFalling : BOOL;
  END_VAR

            
          

METHOD initialize
                  SUPER^.initialize();

lTimer.initialize();
lTimer.Enable := TRUE;

                
END_METHOD

METHOD operator
                  lChanged := (lInput<>lPreviousInput);

lRising := ((lChanged) AND (lInput));
lFalling := ((lChanged) AND (NOT(lInput)));

IF (lRising) THEN
	lTimer.reset();
END_IF

lTimer.operator();
lExpired := ((lInput) AND (lTimer.lExpired));

IF (lFalling) THEN
	lDuration := lTimer.lTimer.ET;
END_IF

lExpiredEvent := FALSE;

// trigger on falling, automatically a one off event
IF (lTriggerOnFalling) THEN
	IF ((lExpired) AND (lFalling)) THEN
		lExpiredEvent := TRUE;
	END_IF

// otherwise require check to ensure one off event
ELSE
	IF ((lExpired) AND (NOT(lExpiredTriggered))) THEN
		lExpiredEvent := lExpiredTriggered := TRUE;
	END_IF
END_IF
	
// reset one off check
IF (NOT(lInput)) THEN
	lExpiredTriggered  := FALSE;
END_IF

// short event that did not last long enough
lFastEvent := FALSE;
IF ((lFalling) AND (NOT(lExpired))) THEN
	lFastEvent := TRUE;
END_IF

lPreviousInput := lInput;
lValue := lExpiredEvent;

SUPER^.operator();

                
END_METHOD

PROPERTY Input : BOOL
SET
                    lInput := Input;
operator();
                  
END_SET
END_PROPERTY

PROPERTY Period : t_time
GET
                    Period := lTimer.Period;
                  
END_GET
SET
                    lTimer.Period := Period;

                  
END_SET
END_PROPERTY
END_FUNCTION_BLOCK

FUNCTION_BLOCK ValueObjectBool EXTENDS ValueObject
  VAR
    lValue : BOOL;
    lOverrideValue : BOOL;
  END_VAR

            
          

METHOD configure
  VAR_INPUT
    executeContext : POINTER TO ExecuteContext;
  END_VAR
                  IF (executeContext^.configureBool(cTokenValue,lValue,FALSE,THIS)) THEN
	RETURN;
END_IF

IF (executeContext^.configureBool(cTokenOverrideValue,lOverrideValue,FALSE,THIS)) THEN
	RETURN;
END_IF

SUPER^.configure(executeContext);


                
END_METHOD

METHOD describe
  VAR_INPUT
    executeContext : POINTER TO ExecuteContext;
  END_VAR
                  SUPER^.describe(executeContext);

IF (executeContext^.matchOption(cExecuteOptionSyntax)) THEN
	executeContext^.describeSyntaxConfigurable(lStyle,cTokenValue,cDataTypeBool,cEnumTypeNone,lUnits,cDescriptionValue);
	executeContext^.describeSyntaxConfigurable(cValueStyleParameter,cTokenOverrideValue,cDataTypeBool,cEnumTypeNone,lUnits,cDescriptionOverrideValue);
	
	RETURN;
END_IF

IF (executeContext^.matchOption(cExecuteOptionParameter)) THEN
	executeContext^.describeParameter(lStyle,lIdentity,cTokenValue,gTypeHandler.getTokenForBool(lValue),cDataTypeBool,cEnumTypeNone,lUnits,cDescriptionValue);
	executeContext^.describeParameter(cValueStyleParameter,lIdentity,cTokenOverrideValue,gTypeHandler.getTokenForBool(lOverrideValue),cDataTypeBool,cEnumTypeNone,lUnits,cDescriptionOverrideValue);
		
	RETURN;
END_IF

executeContext^.appendTokenPair(cTokenValue,gTypeHandler.getTokenForUSINT(BOOL_TO_USINT(lValue)),FALSE,TRUE);
executeContext^.appendTokenPair(cTokenOverrideValue,gTypeHandler.getTokenForUSINT(BOOL_TO_USINT(lOverrideValue)),FALSE,TRUE);


                
END_METHOD

METHOD off
                  lValue := false;
                
END_METHOD

METHOD on
                  lValue := true;
                
END_METHOD

METHOD operator
                  IF (lOverride) THEN
	lValue := lOverrideValue;
END_IF

lCnt := lCnt + 1;

                
END_METHOD

PROPERTY OverrideValue : BOOL
GET
                    OverrideValue := lOverrideValue;
                  
END_GET
SET
                    lOverrideValue := OverrideValue;
                  
END_SET
END_PROPERTY

PROPERTY TypeToken : t_medium_string
GET
                    TypeToken := 'ValObjBool';
                  
END_GET
END_PROPERTY

(* {attribute 'monitoring' := 'call'} *)
PROPERTY Value : BOOL
GET
                    Value := lValue;
                  
END_GET
SET
                    lValue := Value;
                  
END_SET
END_PROPERTY
END_FUNCTION_BLOCK

FUNCTION_BLOCK ValueReferenceBool EXTENDS ValueReference
  VAR
    lValue : REFERENCE TO BOOL;
  END_VAR

            
          

METHOD configure
  VAR_INPUT
    executeContext : POINTER TO ExecuteContext;
  END_VAR
                  IF (executeContext^.configureBool(cTokenValue,lValue,FALSE,THIS)) THEN
	RETURN;
END_IF

SUPER^.configure(executeContext);



                
END_METHOD

METHOD describe
  VAR_INPUT
    executeContext : POINTER TO ExecuteContext;
  END_VAR
                  IF (executeContext^.matchOption(cExecuteOptionParameter)) THEN
	executeContext^.describeParameter(lStyle,lIdentity,cTokenValue,gTypeHandler.getTokenForBool(lValue),cDataTypeBool,cEnumTypeNone,lUnits,cDescriptionValue);	
	RETURN;
END_IF

SUPER^.describe(executeContext);

IF (executeContext^.matchOption(cExecuteOptionSyntax)) THEN
	executeContext^.describeSyntaxConfigurable(lStyle,cTokenValue,cDataTypeBool,cEnumTypeNone,lUnits,cDescriptionValue);
	RETURN;
END_IF

executeContext^.appendTokenPair(cTokenValue,gTypeHandler.getTokenForUSINT(BOOL_TO_USINT(lValue)),FALSE,TRUE);



                
END_METHOD

METHOD initializeValueReference
  VAR_INPUT
    value : REFERENCE TO BOOL;
    p : POINTER TO t_particle_nop;
    _name : t_medium_string;
    description : t_long_string;
    units : t_token_string;
    style : t_value_style;
  END_VAR
                  lValue REF= value;
Name := _name;
Description := description;
lUnits := units;
lStyle := style;

IF (p<>0) THEN
	p^.registerNonOperational(THIS);
END_IF

                
END_METHOD

PROPERTY TypeToken : t_medium_string
GET
                    TypeToken := 'ValRefBool';
                  
END_GET
END_PROPERTY

PROPERTY Value : BOOL
GET
                    Value := lValue;
                  
END_GET
SET
                    lValue := Value;
                  
END_SET
END_PROPERTY
END_FUNCTION_BLOCK

FUNCTION_BLOCK ValueReferencePersistentBool EXTENDS ValueReference
  VAR
    lValue : REFERENCE TO t_persistent_bool;
  END_VAR

            
          

METHOD describe
  VAR_INPUT
    executeContext : POINTER TO ExecuteContext;
  END_VAR
                  IF (executeContext^.matchOption(cExecuteOptionParameter)) THEN
	executeContext^.describeParameter(lStyle,lIdentity,cTokenValue,gTypeHandler.getTokenForBool(lValue.Value),cDataTypeBool,cEnumTypeNone,lUnits,cDescriptionValue);
	RETURN;
END_IF

SUPER^.describe(executeContext);

IF (executeContext^.matchOption(cExecuteOptionSyntax)) THEN
	executeContext^.describeSyntaxConfigurable(lStyle,cTokenValue,cDataTypeBool,cEnumTypeNone,lUnits,cDescriptionValue);
	RETURN;
END_IF

executeContext^.appendTokenPair(cTokenValue,gTypeHandler.getTokenForUSINT(BOOL_TO_USINT(lValue.Value)),FALSE,TRUE);




                
END_METHOD

METHOD configure
  VAR_INPUT
    executeContext : POINTER TO ExecuteContext;
  END_VAR
  VAR
    value : BOOL;
  END_VAR
                  IF (executeContext^.configureBool(cTokenValue,value,FALSE,THIS)) THEN
	lValue.Value := value;
	RETURN;
END_IF

SUPER^.configure(executeContext);



                
END_METHOD

METHOD initializeValueReference
  VAR_INPUT
    value : REFERENCE TO t_persistent_bool;
    p : POINTER TO t_particle_nop;
    _name : t_medium_string;
    description : t_long_string;
    units : t_token_string;
    style : t_value_style;
  END_VAR
                  lValue REF= value;
Name := _name;
Description := description;
lUnits := units;
lStyle := style;

IF (p<>0) THEN
	p^.registerNonOperational(THIS);
END_IF

                
END_METHOD

PROPERTY TypeToken : t_medium_string
GET
                    TypeToken := 'ValRefPersBool';
                  
END_GET
END_PROPERTY

PROPERTY Value : BOOL
GET
                    Value := lValue.Value;
                  
END_GET
SET
                    lValue.Value := Value;
                  
END_SET
END_PROPERTY
END_FUNCTION_BLOCK

FUNCTION_BLOCK ValueReferencePersistentDWORD EXTENDS ValueReference
  VAR
    lValue : REFERENCE TO t_persistent_DWORD;
  END_VAR

            
          

METHOD configure
  VAR_INPUT
    executeContext : POINTER TO ExecuteContext;
  END_VAR
  VAR
    value : DWORD;
  END_VAR
                  IF (executeContext^.configureDWORD(cTokenValue,value,FALSE,THIS)) THEN
	lValue.Value := value;
	RETURN;
END_IF

SUPER^.configure(executeContext);

                
END_METHOD

METHOD initializeValueReference
  VAR_INPUT
    value : REFERENCE TO t_persistent_DWORD;
    p : POINTER TO t_particle_nop;
    _name : t_medium_string;
    description : t_long_string;
    units : t_token_string;
    style : t_value_style;
  END_VAR
                  lValue REF= value;
Name := _name;
Description := description;
lUnits := units;
lStyle := style;

IF (p<>0) THEN
	p^.registerNonOperational(THIS);
END_IF

                
END_METHOD

METHOD describe
  VAR_INPUT
    executeContext : POINTER TO ExecuteContext;
  END_VAR
                  IF (executeContext^.matchOption(cExecuteOptionParameter)) THEN
	executeContext^.describeParameter(lStyle,lIdentity,cTokenValue,gTypeHandler.getTokenForDWORD(lValue.Value),cDataTypeDWORD,cEnumTypeNone,lUnits,cDescriptionValue);	
	RETURN;
END_IF

SUPER^.describe(executeContext);

IF (executeContext^.matchOption(cExecuteOptionSyntax)) THEN
	executeContext^.describeSyntaxConfigurable(lStyle,cTokenValue,cDataTypeDWORD,cEnumTypeNone,lUnits,cDescriptionValue);
	RETURN;
END_IF

executeContext^.appendTokenPair(cTokenValue,gTypeHandler.getTokenForDWORD(lValue.Value),FALSE,TRUE);


                
END_METHOD

PROPERTY TypeToken : t_medium_string
GET
                    TypeToken := 'ValRefPersDWORD';
                  
END_GET
END_PROPERTY

PROPERTY Value : DWORD
GET
                    Value := lValue.Value;
                  
END_GET
SET
                    lValue.Value := Value;
                  
END_SET
END_PROPERTY
END_FUNCTION_BLOCK

FUNCTION_BLOCK ValueObjectEnumTypeInputReferenceUINT EXTENDS ValueObjectEnumType
  VAR
    lIndex : USINT := 0;
    lLength : USINT := 16;
    lInputReference : REFERENCE TO UINT;
  END_VAR

            
          

METHOD operator
                  lValue := fExtractBitsFromWord(lInputReference,pStart:=lIndex,pLength:=lLength);

IF (lOverride) THEN
	lValue := lOverrideValue;
END_IF

                
END_METHOD

METHOD initialize
                  IF (NOT(__ISVALIDREF(lInputReference))) THEN
	gCodeErrorHandler(pMessage:=CONCAT('null reference in ',lIdentity));
END_IF

SUPER^.initialize();

                
END_METHOD

PROPERTY InputReference : REFERENCE TO UINT
SET
                    lInputReference REF= InputReference;


                  
END_SET
END_PROPERTY

PROPERTY Index : USINT
GET
                    Index := lIndex;
                  
END_GET
SET
                    lIndex := MIN(Index,15);
                  
END_SET
END_PROPERTY

PROPERTY Length : USINT
GET
                    Length := lLength;
                  
END_GET
SET
                    lLength := MIN(Length,16);
                  
END_SET
END_PROPERTY
END_FUNCTION_BLOCK

FUNCTION_BLOCK ValueObjectEnumTypeInputReferenceUSINT EXTENDS ValueObjectEnumType
  VAR
    lIndex : USINT := 0;
    lLength : USINT := 8;
    lInputReference : REFERENCE TO USINT;
  END_VAR

            
          

METHOD operator
                  lValue := fExtractBits(lInputReference,pStart:=lIndex,pLength:=lLength);

IF (lOverride) THEN
	lValue := lOverrideValue;
END_IF

                
END_METHOD

METHOD initialize
                  IF (NOT(__ISVALIDREF(lInputReference))) THEN
	gCodeErrorHandler(pMessage:=CONCAT('null reference in ',lIdentity));
END_IF

SUPER^.initialize();

                
END_METHOD

PROPERTY InputReference : REFERENCE TO USINT
SET
                    lInputReference REF= InputReference;


                  
END_SET
END_PROPERTY

PROPERTY Index : USINT
GET
                    Index := lIndex;
                  
END_GET
SET
                    lIndex := MIN(Index,7);
                  
END_SET
END_PROPERTY

PROPERTY Length : USINT
GET
                    Length := lLength;
                  
END_GET
SET
                    lLength := MIN(Length,8);
                  
END_SET
END_PROPERTY
END_FUNCTION_BLOCK

FUNCTION_BLOCK ValueObjectEnumTypeOutputReferenceUSINT EXTENDS ValueObjectEnumType
  VAR
    lOutputReference : REFERENCE TO USINT;
    lIndex : USINT := 0;
    lMergeOutput : BOOL := FALSE;
  END_VAR

            
          

METHOD operator
                  SUPER^.operator();

IF (lMergeOutput) THEN
	lOutputReference := fMergeBits(lOutputReference,lValue,pStart:=lIndex);
ELSE
	lOutputReference := fInsertBits(lValue,pStart:=lIndex);
END_IF

                
END_METHOD

METHOD initialize
                  IF (NOT(__ISVALIDREF(lOutputReference))) THEN
	gCodeErrorHandler(pMessage:=CONCAT('null reference in ',lIdentity));
END_IF

SUPER^.initialize();

                
END_METHOD

PROPERTY OutputReference : REFERENCE TO USINT
SET
                    lOutputReference REF= OutputReference;


                  
END_SET
END_PROPERTY

PROPERTY MergeOutput : BOOL
GET
                    MergeOutput := lMergeOutput;
                  
END_GET
SET
                    lMergeOutput := MergeOutput;
                  
END_SET
END_PROPERTY

PROPERTY Index : USINT
GET
                    Index := lIndex;
                  
END_GET
SET
                    lIndex := MIN(Index,7);
                  
END_SET
END_PROPERTY
END_FUNCTION_BLOCK

FUNCTION_BLOCK ValueObjectEnumType EXTENDS ValueObject
  VAR
    lValue : INT := 0;
    lOverrideValue : INT := 0;
    lEnumType : t_enum_type := cEnumTypeNone;
  END_VAR

            
          

METHOD configure
  VAR_INPUT
    executeContext : POINTER TO ExecuteContext;
  END_VAR
                  IF (executeContext^.configureEnum(lEnumType,cTokenValue,lValue,FALSE,THIS)) THEN
	RETURN;
END_IF

IF (executeContext^.configureEnum(lEnumType,cTokenOverrideValue,lOverrideValue,FALSE,THIS)) THEN
	RETURN;
END_IF

SUPER^.configure(executeContext);

                
END_METHOD

METHOD describe
  VAR_INPUT
    executeContext : POINTER TO ExecuteContext;
  END_VAR
                  SUPER^.describe(executeContext);

IF (executeContext^.matchOption(cExecuteOptionSyntax)) THEN
	executeContext^.describeSyntaxConfigurable(lStyle,cTokenValue,cDataTypeEnum,lEnumType,lUnits,cDescriptionValue);
	executeContext^.describeSyntaxConfigurable(cValueStyleParameter,cTokenOverrideValue,cDataTypeEnum,lEnumType,lUnits,cDescriptionOverrideValue);

	RETURN;
END_IF

IF (executeContext^.matchOption(cExecuteOptionParameter)) THEN
	executeContext^.describeParameter(lStyle,lIdentity,cTokenValue,gTypeHandler.getTokenForEnum(lEnumType,lValue),cDataTypeEnum,lEnumType,lUnits,cDescriptionValue);
	executeContext^.describeParameter(cValueStyleParameter,lIdentity,cTokenOverrideValue,gTypeHandler.getTokenForEnum(lEnumType,lOverrideValue),cDataTypeEnum,lEnumType,lUnits,cDescriptionOverrideValue);
	
	RETURN;
END_IF

executeContext^.appendTokenPair(cTokenValueType,gTypeHandler.getTokenForEnumType(lEnumType),TRUE,TRUE);

executeContext^.appendTokenPair(cTokenValue,gTypeHandler.getTokenForINT(lValue),FALSE,TRUE);
executeContext^.appendTokenPair(cTokenMeaning,gTypeHandler.getTokenForEnum(lEnumType,lValue),TRUE,TRUE);

executeContext^.appendTokenPair(cTokenOverrideValue,gTypeHandler.getTokenForINT(lOverrideValue),FALSE,TRUE);
executeContext^.appendTokenPair(cTokenOverrideMeaning,gTypeHandler.getTokenForEnum(lEnumType,lOverrideValue),TRUE,TRUE);

                
END_METHOD

METHOD operator
                  IF (lOverride) THEN
	lValue := lOverrideValue;
END_IF

                
END_METHOD

PROPERTY OverrideValue : INT
GET
                    OverrideValue := lOverrideValue;
                  
END_GET
SET
                    lOverrideValue := OverrideValue;
                  
END_SET
END_PROPERTY

PROPERTY TypeToken : t_medium_string
GET
                    TypeToken := 'ValObjEnum';
                  
END_GET
END_PROPERTY

(* {attribute 'monitoring' := 'call'} *)
PROPERTY Value : INT
GET
                    Value := lValue;
                  
END_GET
SET
                    lValue := Value;
                  
END_SET
END_PROPERTY

PROPERTY EnumType : t_enum_type
GET
                    EnumType := lEnumType;
                  
END_GET
SET
                    lEnumType := EnumType;
                  
END_SET
END_PROPERTY
END_FUNCTION_BLOCK

FUNCTION_BLOCK ValueReferenceEnumType EXTENDS ValueReference
  VAR
    lValue : REFERENCE TO INT;
    lEnumType : t_enum_type := cEnumTypeNone;
  END_VAR

            
          

METHOD configure
  VAR_INPUT
    executeContext : POINTER TO ExecuteContext;
  END_VAR
                  IF (executeContext^.configureEnum(lEnumType,cTokenValue,lValue,FALSE,THIS)) THEN
	RETURN;
END_IF

SUPER^.configure(executeContext);

                
END_METHOD

METHOD describe
  VAR_INPUT
    executeContext : POINTER TO ExecuteContext;
  END_VAR
                  IF (executeContext^.matchOption(cExecuteOptionParameter)) THEN
	executeContext^.describeParameter(lStyle,lIdentity,cTokenValue,gTypeHandler.getTokenForEnum(lEnumType,lValue),cDataTypeEnum,lEnumType,lUnits,cDescriptionValue);
	RETURN;
END_IF

SUPER^.describe(executeContext);

IF (executeContext^.matchOption(cExecuteOptionSyntax)) THEN
	executeContext^.describeSyntaxConfigurable(lStyle,cTokenValue,cDataTypeEnum,lEnumType,lUnits,cDescriptionValue);
	RETURN;
END_IF

executeContext^.appendTokenPair(cTokenValueType,gTypeHandler.getTokenForEnumType(lEnumType),TRUE,TRUE);

executeContext^.appendTokenPair(cTokenValue,gTypeHandler.getTokenForINT(lValue),FALSE,TRUE);
executeContext^.appendTokenPair(cTokenMeaning,gTypeHandler.getTokenForEnum(lEnumType,lValue),TRUE,TRUE);

                
END_METHOD

METHOD initializeValueReference
  VAR_INPUT
    value : REFERENCE TO INT;
    p : POINTER TO t_particle_nop;
    _name : t_medium_string;
    description : t_long_string;
    units : t_token_string;
    enumType : t_enum_type;
    style : t_value_style;
  END_VAR
                  lValue REF= value;
Name := _name;
Description := description;
lUnits := units;
EnumType := enumType;
lStyle := style;

IF (p<>0) THEN
	p^.registerNonOperational(THIS);
END_IF

                
END_METHOD

PROPERTY TypeToken : t_medium_string
GET
                    TypeToken := 'ValRefEnumType';
                  
END_GET
END_PROPERTY

PROPERTY Value : INT
GET
                    Value := lValue;
                  
END_GET
SET
                    lValue := Value;
                  
END_SET
END_PROPERTY

PROPERTY EnumType : t_enum_type
GET
                    EnumType := lEnumType;
                  
END_GET
SET
                    lEnumType := EnumType;
                  
END_SET
END_PROPERTY
END_FUNCTION_BLOCK

FUNCTION_BLOCK ValueObjectPercentageCurve EXTENDS ValueObjectPercentageSmooth
  VAR
    lPrevious : t_percentage;
    lDeltaPrevious : t_percentage;
    lDelta : t_percentage;
    lNonZero : t_percentage;
    lNonZeroPrevious : t_percentage;
    lEquivalentThreshold : t_percentage := 0.0;
    lInflexions : USINT;
    lResetFlag : BOOL := FALSE;
  END_VAR

            
          

METHOD operator
  VAR
    percInput : REAL;
  END_VAR
                  lPrevious := lValue;
lResetFlag := FALSE;

SUPER^.operator();

lDeltaPrevious := lDelta;
IF (ABS(lValue-lPrevious)>=lEquivalentThreshold) THEN
	lDelta := lValue - lPrevious;
END_IF

lNonZeroPrevious := lNonZero;
IF (ABS(lValue)>=lEquivalentThreshold) THEN
	lNonZero := lValue;
END_IF

IF (((lDeltaPrevious<0.0) AND (lDelta>0.0)) OR
	((lDeltaPrevious>0.0) AND (lDelta<0.0)) OR
	((lNonZeroPrevious<0.0) AND (lNonZero>0.0)) OR
	((lNonZeroPrevious>0.0) AND (lNonZero<0.0))) THEN
	lInflexions := lInflexions + 1;
END_IF

                
END_METHOD

METHOD reset
                  lInflexions := 0;
	//lMovementCount := 0;
	//lRequestedDelta := 0.0;
	//lRequestedDeltaPrevious := 0.0;
	
lDelta := 0.0;
lDeltaPrevious := 0.0;

lResetFlag := TRUE;

                
END_METHOD

PROPERTY Inflexions : USINT
GET
                    Inflexions := lInflexions;
                  
END_GET
END_PROPERTY
END_FUNCTION_BLOCK

FUNCTION_BLOCK ValueObjectPercentageInputAsSINT EXTENDS ValueObjectPercentage
  VAR
    lInput : SINT;
  END_VAR

            
          

METHOD operator
                  lValue := SINT_TO_REAL(lInput)/127.0;

SUPER^.operator();

                
END_METHOD

PROPERTY Input : SINT
SET
                    lInput := Input;
operator();

                  
END_SET
END_PROPERTY
END_FUNCTION_BLOCK

FUNCTION_BLOCK ValueObjectPercentageInputReferenceByte EXTENDS ValueObjectPercentage
  VAR
    lInputReference : REFERENCE TO BYTE;
  END_VAR

            
          

METHOD operator
                  lValue := SINT_TO_REAL(BYTE_TO_SINT(lInputReference))/127.0;

SUPER^.operator();


                
END_METHOD

METHOD initialize
                  IF (NOT(__ISVALIDREF(lInputReference))) THEN
	gCodeErrorHandler(pMessage:=CONCAT('null reference in ',lIdentity));
END_IF

SUPER^.initialize();

                
END_METHOD

PROPERTY InputReference : REFERENCE TO BYTE
SET
                    lInputReference REF= InputReference;


                  
END_SET
END_PROPERTY
END_FUNCTION_BLOCK

FUNCTION_BLOCK ValueObjectPercentageInputReferenceINTJoystick EXTENDS ValueObjectPercentageSmooth
  VAR CONSTANT
    cJoystickLimit : INT := 32000;
    cValueThreshold : t_percentage := 0.025;
  END_VAR
  VAR
    lInputReference : REFERENCE TO INT;
    lFactor : REAL := 1.0;
    lPower : REAL := 1.0;
    lDeadband : INT := 1000;
    lValueThreshold : t_percentage := cValueThreshold;
  END_VAR

            
          

METHOD operator
                  IF (lInputReference>lDeadband) THEN
	lInputAsPercentage := INT_TO_REAL(lInputReference-lDeadband)/INT_TO_REAL(cJoystickLimit-lDeadband);
	lInputAsPercentage := EXPT(lInputAsPercentage,lPower);
ELSIF (lInputReference<(0-lDeadband)) THEN
	lInputAsPercentage := INT_TO_REAL(lInputReference+lDeadband)/INT_TO_REAL(cJoystickLimit-lDeadband);
	lInputAsPercentage := EXPT(ABS(lInputAsPercentage),lPower)*(-1.0);
ELSE
	lInputAsPercentage := 0.0;
END_IF

SUPER^.operator();

IF (lValue>0) THEN
	lValue := MIN(lValue * lFactor,1.0);
END_IF
IF (lValue<0) THEN
	lValue := MAX(lValue * lFactor,-1.0);
END_IF

IF (ABS(lValue)<lValueThreshold) THEN
	lValue := 0.0;
END_IF

                
END_METHOD

METHOD initialize
                  IF (NOT(__ISVALIDREF(lInputReference))) THEN
	gCodeErrorHandler(pMessage:=CONCAT('null reference in ',lIdentity));
END_IF

SUPER^.initialize();

                
END_METHOD

PROPERTY Power : REAL
GET
                    Power := lPower;
                  
END_GET
SET
                    lPower := ABS(Power);

                  
END_SET
END_PROPERTY

PROPERTY Deadband : INT
GET
                    Deadband := lDeadband;
                  
END_GET
SET
                    lDeadband := ABS(Deadband);

                  
END_SET
END_PROPERTY

PROPERTY Factor : REAL
GET
                    Factor := lFactor;
                  
END_GET
SET
                    lFactor := ABS(Factor);

                  
END_SET
END_PROPERTY

PROPERTY InputPresent : BOOL
GET
                    InputPresent := (lInputAsPercentage<>0.0);
                  
END_GET
END_PROPERTY

PROPERTY ValueThreshold : t_percentage
GET
                    ValueThreshold := lValueThreshold;
                  
END_GET
SET
                    lValueThreshold := ValueThreshold;
                  
END_SET
END_PROPERTY

PROPERTY InputReference : REFERENCE TO INT
SET
                    lInputReference REF= InputReference;


                  
END_SET
END_PROPERTY
END_FUNCTION_BLOCK

FUNCTION_BLOCK ValueObjectPercentageInputReferenceSINT EXTENDS ValueObjectRealScaledOffset
  VAR
    lInputReference : REFERENCE TO SINT;
  END_VAR

            
          

METHOD operator
                  lValue := SINT_TO_REAL(lInputReference)/127.0;

SUPER^.operator();


                
END_METHOD

METHOD initialize
                  IF (NOT(__ISVALIDREF(lInputReference))) THEN
	gCodeErrorHandler(pMessage:=CONCAT('null reference in ',lIdentity));
END_IF

SUPER^.initialize();

                
END_METHOD

PROPERTY InputReference : REFERENCE TO SINT
SET
                    lInputReference REF= InputReference;


                  
END_SET
END_PROPERTY
END_FUNCTION_BLOCK

FUNCTION_BLOCK ValueObjectPercentageInputReferenceUSINTJoystick EXTENDS ValueObjectPercentageSmooth
  VAR
    lInputReference : REFERENCE TO USINT;
    lFactor : REAL := 1.0;
    lPower : REAL := 1.0;
    lDeadband : USINT := 5;
  END_VAR

            
          

METHOD operator
  VAR
    percInput : REAL;
  END_VAR
                  IF (lInputReference>(128+lDeadband)) THEN
	lInputAsPercentage := USINT_TO_REAL(lInputReference-128-lDeadband)/USINT_TO_REAL(127-lDeadband);
ELSIF (lInputReference<(128-lDeadband)) THEN
	lInputAsPercentage := 0.0 - USINT_TO_REAL(128-lDeadband-lInputReference)/USINT_TO_REAL(128-lDeadband);
ELSE
	lInputAsPercentage := 0.0;
END_IF

lInputAsPercentage := EXPT(lInputAsPercentage,lPower);

SUPER^.operator();

IF (lValue>0) THEN
	lValue := MIN(lValue * lFactor,1.0);
END_IF
IF (lValue<0) THEN
	lValue := MAX(lValue * lFactor,-1.0);
END_IF

                
END_METHOD

METHOD initialize
                  IF (NOT(__ISVALIDREF(lInputReference))) THEN
	gCodeErrorHandler(pMessage:=CONCAT('null reference in ',lIdentity));
END_IF

SUPER^.initialize();

                
END_METHOD

PROPERTY Deadband : USINT
GET
                    Deadband := lDeadband;
                  
END_GET
SET
                    lDeadband := ABS(Deadband);

                  
END_SET
END_PROPERTY

PROPERTY Factor : REAL
GET
                    Factor := lFactor;
                  
END_GET
SET
                    lFactor := ABS(Factor);

                  
END_SET
END_PROPERTY

PROPERTY InputPresent : BOOL
GET
                    InputPresent := (lInputAsPercentage<>0.0);
                  
END_GET
END_PROPERTY

PROPERTY Power : REAL
GET
                    Power := lPower;
                  
END_GET
SET
                    lPower := ABS(Power);

                  
END_SET
END_PROPERTY

PROPERTY InputReference : REFERENCE TO USINT
SET
                    lInputReference REF= InputReference;


                  
END_SET
END_PROPERTY
END_FUNCTION_BLOCK

FUNCTION_BLOCK ValueObjectPercentageOutputReferenceSINT EXTENDS ValueObjectPercentage
  VAR
    lOutputReference : REFERENCE TO SINT;
  END_VAR

            
          

METHOD operator
                  SUPER^.operator();

lOutputReference := REAL_TO_SINT(MIN(MAX(-127,(lValue*127.0)),127));

                
END_METHOD

METHOD initialize
                  IF (NOT(__ISVALIDREF(lOutputReference))) THEN
	gCodeErrorHandler(pMessage:=CONCAT('null reference in ',lIdentity));
END_IF

SUPER^.initialize();

                
END_METHOD

PROPERTY OutputReference : REFERENCE TO SINT
SET
                    lOutputReference ref= OutputReference;
                  
END_SET
END_PROPERTY
END_FUNCTION_BLOCK

FUNCTION_BLOCK ValueObjectPercentageOutputReferenceUSINT EXTENDS ValueObjectPercentage
  VAR
    lOutputReference : REFERENCE TO USINT;
  END_VAR

            
          

METHOD operator
                  SUPER^.operator();

lOutputReference := REAL_TO_USINT(MIN(MAX(0,(lValue*128.0)+128),255));

                
END_METHOD

METHOD initialize
                  IF (NOT(__ISVALIDREF(lOutputReference))) THEN
	gCodeErrorHandler(pMessage:=CONCAT('null reference in ',lIdentity));
END_IF

SUPER^.initialize();

                
END_METHOD

PROPERTY OutputReference : REFERENCE TO USINT
SET
                    lOutputReference ref= OutputReference;
                  
END_SET
END_PROPERTY
END_FUNCTION_BLOCK

FUNCTION_BLOCK ValueObjectPercentageScaledOffset EXTENDS ValueObjectPercentage
  VAR
    lScaling : REAL := 1.0;
    lOffset : REAL := 0.0;
  END_VAR

            
          

PROPERTY Offset : REAL
GET
                    Offset := lOffset;
                  
END_GET
SET
                    lOffset := Offset;
                  
END_SET
END_PROPERTY

PROPERTY Scaling : REAL
GET
                    Scaling := lScaling;
                  
END_GET
SET
                    lScaling := Scaling;
                  
END_SET
END_PROPERTY
END_FUNCTION_BLOCK

FUNCTION_BLOCK ValueObjectPercentageScaledOffsetInputReferenceUSINT EXTENDS ValueObjectPercentageScaledOffset
  VAR
    lInputReference : REFERENCE TO USINT;
  END_VAR

            
          

METHOD operator
                  lValue := (USINT_TO_REAL(lInputReference)*lScaling)+lOffset;

SUPER^.operator();


                
END_METHOD

METHOD initialize
                  IF (NOT(__ISVALIDREF(lInputReference))) THEN
	gCodeErrorHandler(pMessage:=CONCAT('null reference in ',lIdentity));
END_IF

SUPER^.initialize();

                
END_METHOD

PROPERTY InputReference : REFERENCE TO USINT
SET
                    lInputReference REF= InputReference;


                  
END_SET
END_PROPERTY
END_FUNCTION_BLOCK

FUNCTION_BLOCK ValueObjectPercentageScaledOffsetInputUSINT EXTENDS ValueObjectPercentageScaledOffset
  VAR
    lInput : USINT;
  END_VAR

            
          

METHOD operator
                  lValue := (USINT_TO_REAL(lInput)*lScaling)+lOffset;

SUPER^.operator();


                
END_METHOD

PROPERTY Input : USINT
SET
                    lInput := Input;
operator();

                  
END_SET
END_PROPERTY
END_FUNCTION_BLOCK

FUNCTION_BLOCK ValueObjectPercentageScaledOffsetOutputPercentageNP EXTENDS ValueObjectPercentageScaledOffset
  VAR
    lOutput : t_percentage;
  END_VAR

            
          

METHOD operator
                  SUPER^.operator();

lOutput := (lValue*lScaling)+lOffset;
lOutput := MAX(MIN(lOutput,1.0),-1.0);

                
END_METHOD
END_FUNCTION_BLOCK

FUNCTION_BLOCK ValueObjectPercentageScaledOffsetOutputReferenceINT EXTENDS ValueObjectPercentageScaledOffset
  VAR
    lOutputReference : REFERENCE TO INT;
  END_VAR

            
          

METHOD operator
                  SUPER^.operator();

lOutputReference := REAL_TO_INT((ABS(lValue)*lScaling)+lOffset);

                
END_METHOD

METHOD initialize
                  IF (NOT(__ISVALIDREF(lOutputReference))) THEN
	gCodeErrorHandler(pMessage:=CONCAT('null reference in ',lIdentity));
END_IF

SUPER^.initialize();

                
END_METHOD

PROPERTY OutputReference : REFERENCE TO INT
SET
                    lOutputReference ref= OutputReference;
                  
END_SET
END_PROPERTY
END_FUNCTION_BLOCK

FUNCTION_BLOCK ValueObjectPercentageScaledOffsetOutputReferenceINTChecks EXTENDS ValueObjectPercentageScaledOffsetOutputReferenceINT
  VAR
    lReportedReference : REFERENCE TO INT;
    lFeedbackReference : REFERENCE TO INT;
    lDelta : INT;
    lAlarm : ReportableAlarm;
  END_VAR

            
          

METHOD operator
                  SUPER^.operator();

lDelta := ABS(lOutputReference-lFeedbackReference);

//foobar error handling



                
END_METHOD

METHOD initialize
                  IF ((NOT(__ISVALIDREF(lReportedReference))) OR
	(NOT(__ISVALIDREF(lFeedbackReference)))) THEN
	gCodeErrorHandler(pMessage:=CONCAT('null reference in ',lIdentity));
END_IF

lAlarm.Code := cACOutputFailure;
lAlarm.Name := getStringForStateCode(lAlarm.Code);
lAlarm.Parent:= THIS;

SUPER^.initialize();

lAlarm.initialize();


                
END_METHOD

METHOD getParticle : POINTER TO t_particle
  VAR_INPUT
    name : REFERENCE TO t_token_string;
    id : t_particle_id;
  END_VAR
                  IF (strcmp(name,lAlarm.lName)) THEN
	getParticle := ADR(lAlarm);
	RETURN;
END_IF

getParticle := SUPER^.getParticle(name,id);

                
END_METHOD

METHOD recurse
  VAR_INPUT
    executeContext : POINTER TO ExecuteContext;
  END_VAR
  VAR
    i : USINT;
  END_VAR
                  SUPER^.recurse(executeContext);

IF (NOT(executeContext^.matchOption(cExecuteOptionRecurse))) THEN	
	RETURN;
END_IF

lAlarm.recurse(executeContext);

                
END_METHOD

METHOD describe
  VAR_INPUT
    executeContext : POINTER TO ExecuteContext;
  END_VAR
  VAR
    i : USINT;
    comma : BOOL;
  END_VAR
                  SUPER^.describe(executeContext);

IF (executeContext^.matchOption(cExecuteOptionSyntax)) THEN
	RETURN;
END_IF

IF (executeContext^.matchOption(cExecuteOptionParameter)) THEN
	RETURN;
END_IF

IF (NOT(executeContext^.matchOption(cExecuteOptionChildren))) THEN
	RETURN;
END_IF

executeContext^.append(',"alarm": ');
executeContext^.WriteStream^.increaseIndent();

executeContext^.recordInitiatorWithNewlineIndent();
executeContext^.appendPair('identity',lAlarm.lIdentity,TRUE,FALSE);
executeContext^.appendPair('type',lAlarm.TypeToken,TRUE,TRUE);
executeContext^.appendPair('subsystem',gTypeHandler.getTokenForEnum(cEnumTypeSubsystem,lAlarm.SubSystem),TRUE,TRUE);
executeContext^.recordTerminator();

executeContext^.WriteStream^.decreaseIndent();

                
END_METHOD

PROPERTY FeedbackReference : REFERENCE TO INT
SET
                    lFeedbackReference ref= FeedbackReference;
                  
END_SET
END_PROPERTY

PROPERTY ReportedReference : REFERENCE TO INT
SET
                    lReportedReference ref= ReportedReference;
                  
END_SET
END_PROPERTY

PROPERTY Feedback : INT
GET
                    Feedback := lFeedbackReference;
                  
END_GET
END_PROPERTY

PROPERTY Delta : INT
GET
                    Delta := lDelta;
                  
END_GET
END_PROPERTY

PROPERTY Reported : INT
GET
                    Reported := lReportedReference;
                  
END_GET
END_PROPERTY

PROPERTY Off : BOOL
GET
                    Off := (Value=0.0);
                  
END_GET
SET
                    IF (Off) THEN
	Value := 0.0;
ELSE
	Value := 1.0;	
END_IF
                  
END_SET
END_PROPERTY

PROPERTY On : BOOL
GET
                    On := (Value=1.0); //foobar error handling
                  
END_GET
SET
                    IF (On) THEN
	Value := 1.0;
ELSE
	Value := 0.0;	
END_IF
                  
END_SET
END_PROPERTY

PROPERTY OK : BOOL
GET
                    
                  
END_GET
END_PROPERTY
END_FUNCTION_BLOCK

FUNCTION_BLOCK ValueObjectPercentageSmooth EXTENDS ValueObjectPercentage
  VAR
    lInputAsPercentage : t_percentage;
    lAlpha : REAL := 0.6;
  END_VAR

            
          

METHOD operator
  VAR
    percInput : REAL;
  END_VAR
                  //lValue := (lValue*USINT_TO_REAL(lNumberSamples-1) + (USINT_TO_REAL(lInput)/128.0 - 1.0))/(USINT_TO_REAL(lNumberSamples));
lValue := lValue*(1.0-lAlpha) + lInputAsPercentage*lAlpha;

SUPER^.operator();

                
END_METHOD

PROPERTY Alpha : REAL
GET
                    Alpha := lAlpha;
                  
END_GET
SET
                    lAlpha := Alpha;
                  
END_SET
END_PROPERTY

PROPERTY InputAsPercentage : t_percentage
SET
                    lInputAsPercentage := InputAsPercentage;

                  
END_SET
END_PROPERTY
END_FUNCTION_BLOCK

FUNCTION_BLOCK ValueObjectPercentageSmoothConditional EXTENDS ValueObjectPercentage
  VAR
    lInputAsPercentage : t_percentage;
    lPreviousAsPercentage : t_percentage := 0.0;
    lAlpha : REAL := 1.0;
  END_VAR

            
          

METHOD operator
  VAR
    percInput : REAL;
  END_VAR
                  //lValue := (lValue*USINT_TO_REAL(lNumberSamples-1) + (USINT_TO_REAL(lInput)/128.0 - 1.0))/(USINT_TO_REAL(lNumberSamples));
lValue := lPreviousAsPercentage*(1.0-lAlpha) + lInputAsPercentage*lAlpha;

SUPER^.operator();

lPreviousAsPercentage := lValue;

                
END_METHOD

PROPERTY Alpha : REAL
GET
                    Alpha := lAlpha;
                  
END_GET
SET
                    lAlpha := Alpha;
                  
END_SET
END_PROPERTY

PROPERTY InputAsPercentage : t_percentage
SET
                    lInputAsPercentage := InputAsPercentage;

                  
END_SET
END_PROPERTY

PROPERTY PreviousAsPercentage : t_percentage
SET
                    lPreviousAsPercentage := PreviousAsPercentage;

                  
END_SET
END_PROPERTY

(* {attribute 'monitoring' := 'call'} *)
PROPERTY Value : t_percentage
GET
                    Value := lValue;
                  
END_GET
SET
                    lValue := Value;
lInputAsPercentage := Value;
                  
END_SET
END_PROPERTY
END_FUNCTION_BLOCK

FUNCTION_BLOCK ValuePercentageInputUSINT EXTENDS ValueObjectPercentage
  VAR
    lInput : USINT;
  END_VAR

            
          

METHOD operator
                  lValue := USINT_TO_REAL(lInput)/128.0 - 1.0;

SUPER^.operator();

                
END_METHOD
END_FUNCTION_BLOCK

FUNCTION_BLOCK ValuePercentageScaledOffsetOutputUINT EXTENDS ValuePercentageScaledOffset
  VAR
    lOutput : UINT;
  END_VAR

            
          

METHOD operator
                  SUPER^.operator();

lOutput := REAL_TO_UINT((lValue+lOffset)*lScaling);

                
END_METHOD
END_FUNCTION_BLOCK

FUNCTION_BLOCK ValueObjectPercentage EXTENDS ValueObject
  VAR
    lValue : t_percentage := 0.0;
    lOverrideValue : t_percentage;
  END_VAR

            
          

METHOD configure
  VAR_INPUT
    executeContext : POINTER TO ExecuteContext;
  END_VAR
                  IF (executeContext^.configurePercentage(cTokenValue,lValue,FALSE,THIS)) THEN
	RETURN;
END_IF

IF (executeContext^.configurePercentage(cTokenOverrideValue,lOverrideValue,FALSE,this)) THEN
	RETURN;
END_IF

SUPER^.configure(executeContext);


                
END_METHOD

METHOD describe
  VAR_INPUT
    executeContext : POINTER TO ExecuteContext;
  END_VAR
                  SUPER^.describe(executeContext);

IF (executeContext^.matchOption(cExecuteOptionSyntax)) THEN
	executeContext^.describeSyntaxConfigurable(lStyle,cTokenValue,cDataTypePercentage,cEnumTypeNone,lUnits,cDescriptionValue);
	executeContext^.describeSyntaxConfigurable(cValueStyleParameter,cTokenOverrideValue,cDataTypePercentage,cEnumTypeNone,lUnits,cDescriptionOverrideValue);
	
	RETURN;
END_IF

IF (executeContext^.matchOption(cExecuteOptionParameter)) THEN
	executeContext^.describeParameter(lStyle,lIdentity,cTokenValue,gTypeHandler.getTokenForREAL(lValue),cDataTypePercentage,cEnumTypeNone,lUnits,cDescriptionValue);
	executeContext^.describeParameter(cValueStyleParameter,lIdentity,cTokenOverrideValue,gTypeHandler.getTokenForREAL(lOverrideValue),cDataTypePercentage,cEnumTypeNone,lUnits,cDescriptionOverrideValue);
		
	RETURN;
END_IF

executeContext^.appendTokenPair(cTokenValue,gTypeHandler.getTokenForREAL(lValue),FALSE,TRUE);
executeContext^.appendTokenPair(cTokenOverrideValue,gTypeHandler.getTokenForREAL(lOverrideValue),FALSE,TRUE);

                
END_METHOD

METHOD operator
                  IF (lOverride) THEN
	lValue := lOverrideValue;
END_IF


                
END_METHOD

PROPERTY OverrideValue : t_percentage
GET
                    OverrideValue := lOverrideValue;
                  
END_GET
SET
                    lOverrideValue := OverrideValue;
                  
END_SET
END_PROPERTY

PROPERTY TypeToken : t_medium_string
GET
                    TypeToken := 'ValObjPercentage';
                  
END_GET
END_PROPERTY

(* {attribute 'monitoring' := 'call'} *)
PROPERTY Value : t_percentage
GET
                    Value := lValue;
                  
END_GET
SET
                    lValue := Value;
                  
END_SET
END_PROPERTY
END_FUNCTION_BLOCK

FUNCTION_BLOCK ValueReferencePercentage EXTENDS ValueReference
  VAR
    lValue : REFERENCE TO t_percentage;
  END_VAR

            
          

METHOD configure
  VAR_INPUT
    executeContext : POINTER TO ExecuteContext;
  END_VAR
                  IF (executeContext^.configurePercentage(cTokenValue,lValue,FALSE,this)) THEN
	RETURN;
END_IF

SUPER^.configure(executeContext);



                
END_METHOD

METHOD describe
  VAR_INPUT
    executeContext : POINTER TO ExecuteContext;
  END_VAR
                  IF (executeContext^.matchOption(cExecuteOptionParameter)) THEN
	executeContext^.describeParameter(lStyle,lIdentity,cTokenValue,gTypeHandler.getTokenForREAL(lValue),cDataTypePercentage,cEnumTypeNone,lUnits,cDescriptionValue);
	RETURN;
END_IF

SUPER^.describe(executeContext);

IF (executeContext^.matchOption(cExecuteOptionSyntax)) THEN
	executeContext^.describeSyntaxConfigurable(lStyle,cTokenValue,cDataTypePercentage,cEnumTypeNone,lUnits,cDescriptionValue);
	RETURN;
END_IF

executeContext^.appendTokenPair(cTokenValue,gTypeHandler.getTokenForREAL(lValue),FALSE,TRUE);


                
END_METHOD

METHOD initializeValueReference
  VAR_INPUT
    value : REFERENCE TO t_percentage;
    p : POINTER TO t_particle_nop;
    _name : t_medium_string;
    description : t_long_string;
    units : t_token_string;
    style : t_value_style;
  END_VAR
                  lValue REF= value;
Name := _name;
Description := description;
lUnits := units;
lStyle := style;

IF (p<>0) THEN
	p^.registerNonOperational(THIS);
END_IF

                
END_METHOD

PROPERTY TypeToken : t_medium_string
GET
                    TypeToken := 'ValRefPercentage';
                  
END_GET
END_PROPERTY

PROPERTY Value : t_percentage
GET
                    Value := lValue;
                  
END_GET
SET
                    lValue := Value;
                  
END_SET
END_PROPERTY
END_FUNCTION_BLOCK

FUNCTION_BLOCK ValueObjectRealOffsetScaledInputDINTPositive EXTENDS ValueObjectRealScaledOffset
  VAR
    lInput : DINT;
  END_VAR

            
          

METHOD operator
                  lValue := MAX(0.0,(DINT_TO_REAL(lInput)+lOffset)*lScaling);

SUPER^.operator();

                
END_METHOD

PROPERTY Input : DINT
SET
                    lInput := Input;
operator();

                  
END_SET
END_PROPERTY
END_FUNCTION_BLOCK

FUNCTION_BLOCK ValueObjectRealOffsetScaledInputReferenceUDINT EXTENDS ValueObjectRealScaledOffset
  VAR
    lInputReference : REFERENCE TO UDINT;
  END_VAR

            
          

METHOD operator
                  lValue := (UDINT_TO_REAL(lInputReference)+lOffset)*lScaling;

SUPER^.operator();


                
END_METHOD

METHOD initialize
                  IF (NOT(__ISVALIDREF(lInputReference))) THEN
	gCodeErrorHandler(pMessage:=CONCAT('null reference in ',lIdentity));
END_IF

SUPER^.initialize();

                
END_METHOD

PROPERTY InputReference : REFERENCE TO UDINT
SET
                    lInputReference REF= InputReference;


                  
END_SET
END_PROPERTY
END_FUNCTION_BLOCK

FUNCTION_BLOCK ValueObjectRealOffsetScaledInputUDINT EXTENDS ValueObjectRealScaledOffset
  VAR
    lInput : UDINT;
  END_VAR

            
          

METHOD operator
                  lValue := (UDINT_TO_REAL(lInput)+lOffset)*lScaling;

SUPER^.operator();


                
END_METHOD

PROPERTY Input : UDINT
SET
                    lInput := Input;
operator();

                  
END_SET
END_PROPERTY
END_FUNCTION_BLOCK

FUNCTION_BLOCK ValueObjectRealOffsetScaledOffsetInputReferenceDINT EXTENDS ValueObjectRealScaledOffsetOffset
  VAR
    lInputReference : REFERENCE TO DINT;
  END_VAR

            
          

METHOD operator
                  lValue := MAX(((DINT_TO_REAL(lInputReference)+lOffsetA)*lScaling),0.0)+lOffsetB;

SUPER^.operator();


                
END_METHOD

METHOD initialize
                  IF (NOT(__ISVALIDREF(lInputReference))) THEN
	gCodeErrorHandler(pMessage:=CONCAT('null reference in ',lIdentity));
END_IF

SUPER^.initialize();

                
END_METHOD

PROPERTY InputReference : REFERENCE TO DINT
SET
                    lInputReference REF= InputReference;


                  
END_SET
END_PROPERTY
END_FUNCTION_BLOCK

FUNCTION_BLOCK ValueObjectRealOffsetScaledOutputReferenceUINTSwitched EXTENDS ValueObjectRealScaledOffset
  VAR
    lOutputReference : REFERENCE TO UINT;
  END_VAR

            
          

METHOD operator
  VAR
    w : WORD;
    lsb : BYTE;
    msb : BYTE;
  END_VAR
                  SUPER^.operator();

w := UINT_TO_WORD(REAL_TO_UINT((lValue+lOffset)*lScaling));
lsb := WORD_TO_BYTE(w);
msb := WORD_TO_BYTE(SHR(w,8));

lOutputReference := WORD_TO_UINT(BYTE_TO_WORD(msb) OR SHL(BYTE_TO_WORD(lsb),8));

                
END_METHOD

METHOD initialize
                  IF (NOT(__ISVALIDREF(lOutputReference))) THEN
	gCodeErrorHandler(pMessage:=CONCAT('null reference in ',lIdentity));
END_IF

SUPER^.initialize();

                
END_METHOD

PROPERTY OutputReference : REFERENCE TO UINT
SET
                    lOutputReference ref= OutputReference;
                  
END_SET
END_PROPERTY
END_FUNCTION_BLOCK

FUNCTION_BLOCK ValueObjectRealReference3xUSINT EXTENDS ValueObjectReal
  VAR
    lInputReferenceA : REFERENCE TO USINT;
    lInputReferenceB : REFERENCE TO USINT;
    lInputReferenceC : REFERENCE TO USINT;
  END_VAR

            
          

METHOD operator
                  lValue := UDINT_TO_REAL(SHL(USINT_TO_UDINT(lInputReferenceC),16) +
	SHL(USINT_TO_UDINT(lInputReferenceB),8) +
	USINT_TO_UDINT(lInputReferenceA));

SUPER^.operator();


                
END_METHOD

METHOD initialize
                  IF ((NOT(__ISVALIDREF(lInputReferenceA))) OR
	(NOT(__ISVALIDREF(lInputReferenceB))) OR
	(NOT(__ISVALIDREF(lInputReferenceC)))) THEN
	gCodeErrorHandler(pMessage:=CONCAT('null reference in ',lIdentity));
END_IF

SUPER^.initialize();

                
END_METHOD

PROPERTY InputReferenceA : REFERENCE TO USINT
SET
                    lInputReferenceA REF= InputReferenceA;


                  
END_SET
END_PROPERTY

PROPERTY InputReferenceB : REFERENCE TO USINT
SET
                    lInputReferenceB REF= InputReferenceB;


                  
END_SET
END_PROPERTY

PROPERTY InputReferenceC : REFERENCE TO USINT
SET
                    lInputReferenceC REF= InputReferenceC;


                  
END_SET
END_PROPERTY
END_FUNCTION_BLOCK

FUNCTION_BLOCK ValueObjectRealScaledOffset EXTENDS ValueObjectReal
  VAR
    lScaling : REAL := 1.0;
    lOffset : REAL := 0.0;
  END_VAR

            
          

PROPERTY Offset : REAL
GET
                    Offset := lOffset;
                  
END_GET
SET
                    lOffset := Offset;
                  
END_SET
END_PROPERTY

PROPERTY Scaling : REAL
GET
                    Scaling := lScaling;
                  
END_GET
SET
                    lScaling := Scaling;
                  
END_SET
END_PROPERTY
END_FUNCTION_BLOCK

FUNCTION_BLOCK ValueObjectRealScaledOffsetInputINT EXTENDS ValueObjectRealScaledOffset
  VAR
    lInput : INT;
  END_VAR

            
          

METHOD operator
                  lValue := (INT_TO_REAL(lInput)*lScaling)+lOffset;

SUPER^.operator();


                
END_METHOD

PROPERTY Input : INT
SET
                    lInput := Input;
operator();

                  
END_SET
END_PROPERTY
END_FUNCTION_BLOCK

FUNCTION_BLOCK ValueObjectRealScaledOffsetInputReferenceDINT EXTENDS ValueObjectRealScaledOffset
  VAR
    lInputReference : REFERENCE TO DINT;
  END_VAR

            
          

METHOD initialize
                  IF (NOT(__ISVALIDREF(lInputReference))) THEN
	gCodeErrorHandler(pMessage:=CONCAT('null reference in ',lIdentity));
END_IF

SUPER^.initialize();

                
END_METHOD

METHOD operator
                  lValue := (DINT_TO_REAL(lInputReference)*lScaling)+lOffset;

SUPER^.operator();


                
END_METHOD

PROPERTY InputReference : REFERENCE TO DINT
SET
                    lInputReference REF= InputReference;


                  
END_SET
END_PROPERTY
END_FUNCTION_BLOCK

FUNCTION_BLOCK ValueObjectRealScaledOffsetInputReferenceINT EXTENDS ValueObjectRealScaledOffset
  VAR
    lInputReference : REFERENCE TO INT;
  END_VAR

            
          

METHOD operator
                  lValue := (INT_TO_REAL(lInputReference)*lScaling)+lOffset; // foobar offset and scaling switched, need to standardize

SUPER^.operator();

                
END_METHOD

METHOD initialize
                  IF (NOT(__ISVALIDREF(lInputReference))) THEN
	gCodeErrorHandler(pMessage:=CONCAT('null reference in ',lIdentity));
END_IF

SUPER^.initialize();

                
END_METHOD

PROPERTY InputReference : REFERENCE TO INT
SET
                    lInputReference REF= InputReference;


                  
END_SET
END_PROPERTY
END_FUNCTION_BLOCK

FUNCTION_BLOCK ValueObjectRealScaledOffsetInputReferenceSINT EXTENDS ValueObjectRealScaledOffset
  VAR
    lInputReference : REFERENCE TO SINT;
  END_VAR

            
          

METHOD operator
                  lValue := (SINT_TO_REAL(lInputReference)*lScaling)+lOffset;

SUPER^.operator();


                
END_METHOD

METHOD initialize
                  IF (NOT(__ISVALIDREF(lInputReference))) THEN
	gCodeErrorHandler(pMessage:=CONCAT('null reference in ',lIdentity));
END_IF

SUPER^.initialize();

                
END_METHOD

PROPERTY InputReference : REFERENCE TO SINT
SET
                    lInputReference REF= InputReference;


                  
END_SET
END_PROPERTY
END_FUNCTION_BLOCK

FUNCTION_BLOCK ValueObjectRealScaledOffsetInputReferenceUINT EXTENDS ValueObjectRealScaledOffset
  VAR
    lInputReference : REFERENCE TO UINT;
  END_VAR

            
          

METHOD operator
                  lValue := (UINT_TO_REAL(lInputReference)*lScaling)+lOffset;

SUPER^.operator();

                
END_METHOD

METHOD initialize
                  IF (NOT(__ISVALIDREF(lInputReference))) THEN
	gCodeErrorHandler(pMessage:=CONCAT('null reference in ',lIdentity));
END_IF

SUPER^.initialize();

                
END_METHOD

PROPERTY InputReference : REFERENCE TO UINT
SET
                    lInputReference REF= InputReference;


                  
END_SET
END_PROPERTY
END_FUNCTION_BLOCK

FUNCTION_BLOCK ValueObjectRealScaledOffsetInputReferenceUINTSwitched EXTENDS ValueObjectRealScaledOffset
  VAR
    lInputReference : REFERENCE TO UINT;
  END_VAR

            
          

METHOD initialize
                  IF (NOT(__ISVALIDREF(lInputReference))) THEN
	gCodeErrorHandler(pMessage:=CONCAT('null reference in ',lIdentity));
END_IF

SUPER^.initialize();

                
END_METHOD

METHOD operator
  VAR
    w : WORD;
    lsb : BYTE;
    msb : BYTE;
  END_VAR
                  lsb := WORD_TO_BYTE(UINT_TO_WORD(lInputReference));
msb := WORD_TO_BYTE(SHR(UINT_TO_WORD(lInputReference),8));
w := (BYTE_TO_WORD(msb) OR SHL(BYTE_TO_WORD(lsb),8));

lValue := (UINT_TO_REAL(WORD_TO_UINT(w))*lScaling)+lOffset;

SUPER^.operator();

                
END_METHOD

PROPERTY InputReference : REFERENCE TO UINT
SET
                    lInputReference REF= InputReference;


                  
END_SET
END_PROPERTY
END_FUNCTION_BLOCK

FUNCTION_BLOCK ValueObjectRealScaledOffsetInputReferenceUSINT EXTENDS ValueObjectRealScaledOffset
  VAR
    lInputReference : REFERENCE TO USINT;
  END_VAR

            
          

METHOD operator
                  lValue := (USINT_TO_REAL(lInputReference)*lScaling)+lOffset;

SUPER^.operator();

                
END_METHOD

METHOD initialize
                  IF (NOT(__ISVALIDREF(lInputReference))) THEN
	gCodeErrorHandler(pMessage:=CONCAT('null reference in ',lIdentity));
END_IF

SUPER^.initialize();

                
END_METHOD

PROPERTY InputReference : REFERENCE TO USINT
SET
                    lInputReference REF= InputReference;


                  
END_SET
END_PROPERTY
END_FUNCTION_BLOCK

FUNCTION_BLOCK ValueObjectRealScaledOffsetInputUINT EXTENDS ValueObjectRealScaledOffset
  VAR
    lInput : UINT;
  END_VAR

            
          

METHOD operator
                  lValue := (UINT_TO_REAL(lInput)*lScaling)+lOffset;

SUPER^.operator();


                
END_METHOD

PROPERTY Input : UINT
SET
                    lInput := Input;
operator();

                  
END_SET
END_PROPERTY
END_FUNCTION_BLOCK

FUNCTION_BLOCK ValueObjectRealScaledOffsetInputUSINT EXTENDS ValueObjectRealScaledOffset
  VAR
    lInput : USINT;
  END_VAR

            
          

METHOD operator
                  lValue := (USINT_TO_REAL(lInput)*lScaling)+lOffset;

SUPER^.operator();


                
END_METHOD

PROPERTY Input : USINT
SET
                    lInput := Input;
operator();

                  
END_SET
END_PROPERTY
END_FUNCTION_BLOCK

FUNCTION_BLOCK ValueObjectRealScaledOffsetOffset EXTENDS ValueObjectReal
  VAR
    lScaling : REAL := 1.0;
    lOffsetA : REAL := 0.0;
    lOffsetB : REAL := 0.0;
  END_VAR

            
          

PROPERTY OffsetA : REAL
GET
                    OffsetA := lOffsetA;
                  
END_GET
SET
                    lOffsetA := OffsetA;
                  
END_SET
END_PROPERTY

PROPERTY OffsetB : REAL
GET
                    OffsetB := lOffsetB;
                  
END_GET
SET
                    lOffsetB := OffsetB;
                  
END_SET
END_PROPERTY

PROPERTY Scaling : REAL
GET
                    Scaling := lScaling;
                  
END_GET
SET
                    lScaling := Scaling;
                  
END_SET
END_PROPERTY
END_FUNCTION_BLOCK

FUNCTION_BLOCK ValueObjectRealScaledOffsetOutputReferenceUSINT EXTENDS ValueObjectRealScaledOffset
  VAR
    lOutputReference : REFERENCE TO USINT;
  END_VAR

            
          

METHOD operator
                  SUPER^.operator();

lOutputReference := REAL_TO_USINT((lValue+lOffset)*lScaling); //foobar offset and scaling switched, or is always reversed for ouput versus input

                
END_METHOD

METHOD initialize
                  IF (NOT(__ISVALIDREF(lOutputReference))) THEN
	gCodeErrorHandler(pMessage:=CONCAT('null reference in ',lIdentity));
END_IF

SUPER^.initialize();

                
END_METHOD

PROPERTY OutputReference : REFERENCE TO USINT
SET
                    lOutputReference ref= OutputReference;
                  
END_SET
END_PROPERTY
END_FUNCTION_BLOCK

FUNCTION_BLOCK ValueObjectRealScaledOffsetOutputUINT EXTENDS ValueObjectRealScaledOffset
  VAR
    lOutput : UINT;
  END_VAR

            
          

METHOD operator
                  SUPER^.operator();

lOutput := REAL_TO_UINT((lValue*lScaling)+lOffset);

                
END_METHOD

PROPERTY Output : UINT
GET
                    operator();
Output := lOutput;
                  
END_GET
END_PROPERTY
END_FUNCTION_BLOCK

FUNCTION_BLOCK ValueObjectReal EXTENDS ValueObject
  VAR
    lValue : REAL := 0.0;
    lOverrideValue : REAL;
  END_VAR

            
          

METHOD configure
  VAR_INPUT
    executeContext : POINTER TO ExecuteContext;
  END_VAR
                  IF (executeContext^.configureReal(cTokenValue,lValue,FALSE,THIS)) THEN
	RETURN;
END_IF

IF (executeContext^.configureReal(cTokenOverrideValue,lOverrideValue,FALSE,THIS)) THEN
	RETURN;
END_IF

SUPER^.configure(executeContext);


                
END_METHOD

METHOD describe
  VAR_INPUT
    executeContext : POINTER TO ExecuteContext;
  END_VAR
                  SUPER^.describe(executeContext);

IF (executeContext^.matchOption(cExecuteOptionSyntax)) THEN
	executeContext^.describeSyntaxConfigurable(lStyle,cTokenValue,cDataTypeReal,cEnumTypeNone,lUnits,cDescriptionValue);
	executeContext^.describeSyntaxConfigurable(cValueStyleParameter,cTokenOverrideValue,cDataTypeReal,cEnumTypeNone,lUnits,cDescriptionOverrideValue);
	
	RETURN;
END_IF

IF (executeContext^.matchOption(cExecuteOptionParameter)) THEN
	executeContext^.describeParameter(lStyle,lIdentity,cTokenValue,gTypeHandler.getTokenForREAL(lValue),cDataTypeREAL,cEnumTypeNone,lUnits,cDescriptionValue);
	executeContext^.describeParameter(cValueStyleParameter,lIdentity,cTokenOverrideValue,gTypeHandler.getTokenForREAL(lOverrideValue),cDataTypePercentage,cEnumTypeNone,lUnits,cDescriptionOverrideValue);
		
	RETURN;
END_IF

executeContext^.appendTokenPair(cTokenValue,gTypeHandler.getTokenForREAL(lValue),FALSE,TRUE);
executeContext^.appendTokenPair(cTokenOverrideValue,gTypeHandler.getTokenForREAL(lOverrideValue),FALSE,TRUE);

                
END_METHOD

METHOD operator
                  IF (lOverride) THEN
	lValue := lOverrideValue;
END_IF


                
END_METHOD

PROPERTY OverrideValue : REAL
GET
                    OverrideValue := lOverrideValue;
                  
END_GET
SET
                    lOverrideValue := OverrideValue;
                  
END_SET
END_PROPERTY

PROPERTY TypeToken : t_medium_string
GET
                    TypeToken := 'ValObjReal';
                  
END_GET
END_PROPERTY

(* {attribute 'monitoring' := 'call'} *)
PROPERTY Value : REAL
GET
                    Value := lValue;
                  
END_GET
SET
                    lValue := Value;
                  
END_SET
END_PROPERTY
END_FUNCTION_BLOCK

FUNCTION_BLOCK ValueReferencePersistentReal EXTENDS ValueReference
  VAR
    lValue : REFERENCE TO t_persistent_real;
  END_VAR

            
          

METHOD describe
  VAR_INPUT
    executeContext : POINTER TO ExecuteContext;
  END_VAR
                  IF (executeContext^.matchOption(cExecuteOptionParameter)) THEN
	executeContext^.describeParameter(lStyle,lIdentity,cTokenValue,gTypeHandler.getTokenForREAL(lValue.Value),cDataTypeREAL,cEnumTypeNone,lUnits,cDescriptionValue);
	RETURN;
END_IF

SUPER^.describe(executeContext);

IF (executeContext^.matchOption(cExecuteOptionSyntax)) THEN
	executeContext^.describeSyntaxConfigurable(lStyle,cTokenValue,cDataTypeReal,cEnumTypeNone,lUnits,cDescriptionValue);
	RETURN;
END_IF

executeContext^.appendTokenPair(cTokenValue,gTypeHandler.getTokenForREAL(lValue.Value),FALSE,TRUE);


                
END_METHOD

METHOD configure
  VAR_INPUT
    executeContext : POINTER TO ExecuteContext;
  END_VAR
  VAR
    value : REAL;
  END_VAR
                  IF (executeContext^.configureReal(cTokenValue,value,FALSE,THIS)) THEN
	lValue.Value := value;
	RETURN;
END_IF

SUPER^.configure(executeContext);

                
END_METHOD

METHOD initializeValueReference
  VAR_INPUT
    value : REFERENCE TO t_persistent_real;
    p : POINTER TO t_particle_nop;
    _name : t_medium_string;
    description : t_long_string;
    units : t_token_string;
    style : t_value_style;
  END_VAR
                  lValue REF= value;
Name := _name;
Description := description;
lUnits := units;
lStyle := style;

IF (p<>0) THEN
	p^.registerNonOperational(THIS);
END_IF

                
END_METHOD

PROPERTY TypeToken : t_medium_string
GET
                    TypeToken := 'ValRefPersReal';
                  
END_GET
END_PROPERTY

PROPERTY Value : REAL
GET
                    Value := lValue.Value;
                  
END_GET
SET
                    lValue.Value := Value;
                  
END_SET
END_PROPERTY
END_FUNCTION_BLOCK

FUNCTION_BLOCK ValueReferenceReal EXTENDS ValueReference
  VAR
    lValue : REFERENCE TO REAL;
  END_VAR

            
          

METHOD configure
  VAR_INPUT
    executeContext : POINTER TO ExecuteContext;
  END_VAR
                  IF (executeContext^.configureReal(cTokenValue,lValue,FALSE,THIS)) THEN
	RETURN;
END_IF

SUPER^.configure(executeContext);



                
END_METHOD

METHOD describe
  VAR_INPUT
    executeContext : POINTER TO ExecuteContext;
  END_VAR
                  IF (executeContext^.matchOption(cExecuteOptionParameter)) THEN
	executeContext^.describeParameter(lStyle,lIdentity,cTokenValue,gTypeHandler.getTokenForREAL(lValue),cDataTypeREAL,cEnumTypeNone,lUnits,cDescriptionValue);
	RETURN;
END_IF

SUPER^.describe(executeContext);

IF (executeContext^.matchOption(cExecuteOptionSyntax)) THEN
	executeContext^.describeSyntaxConfigurable(lStyle,cTokenValue,cDataTypeReal,cEnumTypeNone,lUnits,cDescriptionValue);
	RETURN;
END_IF

executeContext^.appendTokenPair(cTokenValue,gTypeHandler.getTokenForREAL(lValue),FALSE,TRUE);


                
END_METHOD

METHOD initializeValueReference
  VAR_INPUT
    value : REFERENCE TO REAL;
    p : POINTER TO t_particle_nop;
    _name : t_medium_string;
    description : t_long_string;
    units : t_token_string;
    style : t_value_style;
  END_VAR
                  lValue REF= value;
Name := _name;
Description := description;
lUnits := units;
lStyle := style;

IF (p<>0) THEN
	p^.registerNonOperational(THIS);
END_IF

                
END_METHOD

PROPERTY TypeToken : t_medium_string
GET
                    TypeToken := 'ValRefReal';
                  
END_GET
END_PROPERTY

PROPERTY Value : REAL
GET
                    Value := lValue;
                  
END_GET
SET
                    lValue := Value;
                  
END_SET
END_PROPERTY
END_FUNCTION_BLOCK

FUNCTION_BLOCK ValueReferencePersistentMediumString EXTENDS ValueReference
  VAR
    lValue : REFERENCE TO t_persistent_medium_string;
  END_VAR

            
          

METHOD configure
  VAR_INPUT
    executeContext : POINTER TO ExecuteContext;
  END_VAR
  VAR
    value : t_medium_string;
  END_VAR
                  IF (executeContext^.configureMediumString(cTokenValue,value,FALSE,THIS)) THEN
	lValue.Value := value;
	RETURN;
END_IF

SUPER^.configure(executeContext);

                
END_METHOD

METHOD initializeValueReference
  VAR_INPUT
    value : REFERENCE TO t_persistent_medium_string;
    p : POINTER TO t_particle_nop;
    _name : t_medium_string;
    description : t_long_string;
    units : t_token_string;
    style : t_value_style;
  END_VAR
                  lValue REF= value;
Name := _name;
Description := description;
lUnits := units;
lStyle := style;

IF (p<>0) THEN
	p^.registerNonOperational(THIS);
END_IF

                
END_METHOD

METHOD describe
  VAR_INPUT
    executeContext : POINTER TO ExecuteContext;
  END_VAR
                  IF (executeContext^.matchOption(cExecuteOptionParameter)) THEN
	executeContext^.describeParameter(lStyle,lIdentity,cTokenValue,lValue.Value,cDataTypeString,cEnumTypeNone,lUnits,cDescriptionValue);
	RETURN;
END_IF

SUPER^.describe(executeContext);

IF (executeContext^.matchOption(cExecuteOptionSyntax)) THEN
	executeContext^.describeSyntaxConfigurable(lStyle,cTokenValue,cDataTypeString,cEnumTypeNone,lUnits,cDescriptionValue);
	RETURN;
END_IF

executeContext^.appendTokenPair(cTokenValue,lValue.Value,TRUE,TRUE);

                
END_METHOD

PROPERTY Value : t_medium_string
GET
                    Value := lValue.Value;
                  
END_GET
SET
                    lValue.Value := Value;
                  
END_SET
END_PROPERTY

PROPERTY TypeToken : t_medium_string
GET
                    TypeToken := 'ValRefPersString';
                  
END_GET
END_PROPERTY
END_FUNCTION_BLOCK

